LIN {X 0,Y 312.499,Z 218.851,A -85,B 0,C 180,E1 -15693.692,E2 -15693.692} C_VEL
LIN {X 0,Y 312.5,Z 218.867,A -85,B 0,C 180,E1 -15697.39,E2 -15697.39} C_VEL
LIN {X 0,Y 312.472,Z 218.863,A -85,B 0,C 180,E1 -15700.713,E2 -15700.713} C_VEL
LIN {X 0,Y 312.435,Z 218.864,A -85,B 0,C 180,E1 -15704.214,E2 -15704.214} C_VEL
LIN {X 0,Y 312.468,Z 218.877,A -85,B 0,C 180,E1 -15707.923,E2 -15707.923} C_VEL
LIN {X 0,Y 312.464,Z 218.86,A -85,B 0,C 180,E1 -15710.972,E2 -15710.972} C_VEL
LIN {X 0,Y 312.52,Z 218.86,A -85,B 0,C 180,E1 -15714.224,E2 -15714.224} C_VEL
LIN {X 0,Y 312.492,Z 218.871,A -85,B 0,C 180,E1 -15717.338,E2 -15717.338} C_VEL
LIN {X 0,Y 312.5,Z 218.867,A -85,B 0,C 180,E1 -15721.296,E2 -15721.296} C_VEL
LIN {X 0,Y 312.541,Z 218.857,A -85,B 0,C 180,E1 -15724.712,E2 -15724.712} C_VEL
LIN {X 0,Y 312.52,Z 218.87,A -85,B 0,C 180,E1 -15728.916,E2 -15728.916} C_VEL
LIN {X 0,Y 312.56,Z 218.863,A -85,B 0,C 180,E1 -15731.261,E2 -15731.261} C_VEL
LIN {X 0,Y 313.478,Z 221.573,A -85,B 0,C 180,E1 -15731.502,E2 -15731.502} C_VEL
LIN {X 0,Y 315.576,Z 224.258,A -85,B 0,C 180,E1 -15731.935,E2 -15731.935} C_VEL
LIN {X 0,Y 317.795,Z 227.6,A -85,B 0,C 180,E1 -15732.4,E2 -15732.4} C_VEL
LIN {X 0,Y 327.062,Z 241.726,A -85,B 0,C 180,E1 -15734.245,E2 -15734.245} C_VEL
LIN {X 0,Y 337.694,Z 259.213,A -85,B 0,C 180,E1 -15736.243,E2 -15736.243} C_VEL
LIN {X 0,Y 345.227,Z 274.119,A -85,B 0,C 180,E1 -15737.624,E2 -15737.624} C_VEL
LIN {X 0,Y 346.756,Z 277.46,A -85,B 0,C 180,E1 -15737.905,E2 -15737.905} C_VEL
LIN {X 0,Y 340.957,Z 418.481,A -85,B 0,C 180,E1 -15740.961,E2 -15740.961} C_VEL
LIN {X 0,Y 339.666,Z 435.003,A -85,B 0,C 180,E1 -15741.526,E2 -15741.526} C_VEL
LIN {X 0,Y 337.912,Z 451.285,A -85,B 0,C 180,E1 -15742.309,E2 -15742.309} C_VEL
LIN {X 0,Y 335.803,Z 467.163,A -85,B 0,C 180,E1 -15743.318,E2 -15743.318} C_VEL
LIN {X 0,Y 333.363,Z 482.624,A -85,B 0,C 180,E1 -15744.559,E2 -15744.559} C_VEL
LIN {X 0,Y 330.649,Z 497.357,A -85,B 0,C 180,E1 -15746.014,E2 -15746.014} C_VEL
LIN {X 0,Y 327.769,Z 511.318,A -85,B 0,C 180,E1 -15747.699,E2 -15747.699} C_VEL
LIN {X 0,Y 325.107,Z 523.063,A -85,B 0,C 180,E1 -15749.384,E2 -15749.384} C_VEL
LIN {X 0,Y 322.619,Z 534.15,A -85,B 0,C 180,E1 -15751.251,E2 -15751.251} C_VEL
LIN {X 0,Y 319.935,Z 545.24,A -85,B 0,C 180,E1 -15753.466,E2 -15753.466} C_VEL
LIN {X 0,Y 317.551,Z 555.075,A -85,B 0,C 180,E1 -15755.813,E2 -15755.813} C_VEL
LIN {X 0,Y 315.438,Z 563.917,A -85,B 0,C 180,E1 -15758.33,E2 -15758.33} C_VEL
LIN {X 0,Y 313.784,Z 571.615,A -85,B 0,C 180,E1 -15760.978,E2 -15760.978} C_VEL
LIN {X 0,Y 312.529,Z 577.931,A -85,B 0,C 180,E1 -15763.66,E2 -15763.66} C_VEL
LIN {X 0,Y 311.627,Z 583.014,A -85,B 0,C 180,E1 -15766.377,E2 -15766.377} C_VEL
LIN {X 0,Y 311.151,Z 586.089,A -85,B 0,C 180,E1 -15768.437,E2 -15768.437} C_VEL
LIN {X 0,Y 310.646,Z 589.194,A -85,B 0,C 180,E1 -15771.224,E2 -15771.224} C_VEL
LIN {X 0,Y 310.372,Z 591.225,A -85,B 0,C 180,E1 -15774.056,E2 -15774.056} C_VEL
LIN {X 0,Y 310.342,Z 592.031,A -85,B 0,C 180,E1 -15776.933,E2 -15776.933} C_VEL
LIN {X 0,Y 310.449,Z 591.683,A -85,B 0,C 180,E1 -15779.873,E2 -15779.873} C_VEL
LIN {X 0,Y 310.685,Z 590.096,A -85,B 0,C 180,E1 -15782.884,E2 -15782.884} C_VEL
LIN {X 0,Y 311.169,Z 587.504,A -85,B 0,C 180,E1 -15785.6,E2 -15785.6} C_VEL
LIN {X 0,Y 311.823,Z 584.455,A -85,B 0,C 180,E1 -15787.921,E2 -15787.921} C_VEL
LIN {X 0,Y 312.836,Z 579.795,A -85,B 0,C 180,E1 -15790.621,E2 -15790.621} C_VEL
LIN {X 0,Y 312.66,Z 577.864,A -85,B 0,C 180,E1 -15791.643,E2 -15791.643} C_VEL
LIN {X 0,Y 310.678,Z 574.56,A -85,B 0,C 180,E1 -15793.323,E2 -15793.323} C_VEL
LIN {X 0,Y 308.852,Z 570.931,A -85,B 0,C 180,E1 -15794.998,E2 -15794.998} C_VEL
LIN {X 0,Y 308.926,Z 568.371,A -85,B 0,C 180,E1 -15795.991,E2 -15795.991} C_VEL
LIN {X 0,Y 311.415,Z 559.856,A -85,B 0,C 180,E1 -15798.719,E2 -15798.719} C_VEL
LIN {X 0,Y 314.117,Z 550.493,A -85,B 0,C 180,E1 -15801.209,E2 -15801.209} C_VEL
LIN {X 0,Y 317.096,Z 540.388,A -85,B 0,C 180,E1 -15803.46,E2 -15803.46} C_VEL
LIN {X 0,Y 320.339,Z 528.936,A -85,B 0,C 180,E1 -15805.596,E2 -15805.596} C_VEL
LIN {X 0,Y 323.619,Z 516.635,A -85,B 0,C 180,E1 -15807.515,E2 -15807.515} C_VEL
LIN {X 0,Y 327.011,Z 503.039,A -85,B 0,C 180,E1 -15809.281,E2 -15809.281} C_VEL
LIN {X 0,Y 330.189,Z 489.128,A -85,B 0,C 180,E1 -15810.773,E2 -15810.773} C_VEL
LIN {X 0,Y 333.066,Z 474.376,A -85,B 0,C 180,E1 -15812.082,E2 -15812.082} C_VEL
LIN {X 0,Y 335.817,Z 458.032,A -85,B 0,C 180,E1 -15813.218,E2 -15813.218} C_VEL
LIN {X 0,Y 337.97,Z 441.536,A -85,B 0,C 180,E1 -15814.106,E2 -15814.106} C_VEL
LIN {X 0,Y 339.513,Z 426.232,A -85,B 0,C 180,E1 -15814.707,E2 -15814.707} C_VEL
LIN {X 0,Y 340.683,Z 408.213,A -85,B 0,C 180,E1 -15815.189,E2 -15815.189} C_VEL
LIN {X 0,Y 346.82,Z 283.058,A -85,B 0,C 180,E1 -15817.956,E2 -15817.956} C_VEL
LIN {X 0,Y 340.843,Z 271.151,A -85,B 0,C 180,E1 -15819.35,E2 -15819.35} C_VEL
LIN {X 0,Y 335.608,Z 261.937,A -85,B 0,C 180,E1 -15820.612,E2 -15820.612} C_VEL
LIN {X 0,Y 328.374,Z 250.883,A -85,B 0,C 180,E1 -15822.45,E2 -15822.45} C_VEL
LIN {X 0,Y 322.618,Z 242.69,A -85,B 0,C 180,E1 -15824.028,E2 -15824.028} C_VEL
LIN {X 0,Y 320.08,Z 239.215,A -85,B 0,C 180,E1 -15824.762,E2 -15824.762} C_VEL
LIN {X 0,Y 316.654,Z 234.675,A -85,B 0,C 180,E1 -15825.796,E2 -15825.796} C_VEL
LIN {X 0,Y 314.086,Z 231.193,A -85,B 0,C 180,E1 -15826.617,E2 -15826.617} C_VEL
LIN {X 0,Y 313.539,Z 230.399,A -85,B 0,C 180,E1 -15826.799,E2 -15826.799} C_VEL
LIN {X 0,Y 311.036,Z 227.861,A -85,B 0,C 180,E1 -15827.604,E2 -15827.604} C_VEL
LIN {X 0,Y 309.624,Z 225.269,A -85,B 0,C 180,E1 -15828.129,E2 -15828.129} C_VEL
LIN {X 0,Y 307.205,Z 223.361,A -85,B 0,C 180,E1 -15828.953,E2 -15828.953} C_VEL
LIN {X 0,Y 305.962,Z 221.144,A -85,B 0,C 180,E1 -15829.452,E2 -15829.452} C_VEL
LIN {X 0,Y 305.646,Z 219.722,A -85,B 0,C 180,E1 -15829.65,E2 -15829.65} C_VEL
LIN {X 0,Y 305.844,Z 219.698,A -85,B 0,C 180,E1 -15833.402,E2 -15833.402} C_VEL
LIN {X 0,Y 305.958,Z 219.681,A -85,B 0,C 180,E1 -15838.683,E2 -15838.683} C_VEL
LIN {X 0,Y 305.958,Z 219.681,A -85,B 0,C 180,E1 -15841.316,E2 -15841.316} C_VEL
LIN {X 0,Y 305.677,Z 219.717,A -85,B 0,C 180,E1 -15845.276,E2 -15845.276} C_VEL
LIN {X 0,Y 305.767,Z 219.705,A -85,B 0,C 180,E1 -15847.926,E2 -15847.926} C_VEL
LIN {X 0,Y 305.601,Z 219.731,A -85,B 0,C 180,E1 -15851.945,E2 -15851.945} C_VEL
LIN {X 0,Y 305.612,Z 219.729,A -85,B 0,C 180,E1 -15855.013,E2 -15855.013} C_VEL
LIN {X 0,Y 305.521,Z 219.734,A -85,B 0,C 180,E1 -15858.786,E2 -15858.786} C_VEL
LIN {X 0,Y 305.491,Z 219.745,A -85,B 0,C 180,E1 -15863.038,E2 -15863.038} C_VEL
LIN {X 0,Y 305.535,Z 219.737,A -85,B 0,C 180,E1 -15866.219,E2 -15866.219} C_VEL
LIN {X 0,Y 305.484,Z 219.742,A -85,B 0,C 180,E1 -15869.043,E2 -15869.043} C_VEL
LIN {X 0,Y 305.468,Z 219.746,A -85,B 0,C 180,E1 -15873.516,E2 -15873.516} C_VEL
LIN {X 0,Y 305.513,Z 219.832,A -85,B 0,C 180,E1 -15875.788,E2 -15875.788} C_VEL
LIN {X 0,Y 306.147,Z 222.012,A -85,B 0,C 180,E1 -15876.645,E2 -15876.645} C_VEL
LIN {X 0,Y 307.4,Z 224.338,A -85,B 0,C 180,E1 -15877.703,E2 -15877.703} C_VEL
LIN {X 0,Y 309.267,Z 227.241,A -85,B 0,C 180,E1 -15878.492,E2 -15878.492} C_VEL
LIN {X 0,Y 313.704,Z 233.179,A -85,B 0,C 180,E1 -15880,E2 -15880} C_VEL
LIN {X 0,Y 317.317,Z 238.242,A -85,B 0,C 180,E1 -15881.152,E2 -15881.152} C_VEL
LIN {X 0,Y 321.927,Z 245.16,A -85,B 0,C 180,E1 -15882.542,E2 -15882.542} C_VEL
LIN {X 0,Y 327.398,Z 253.587,A -85,B 0,C 180,E1 -15884.077,E2 -15884.077} C_VEL
LIN {X 0,Y 335.467,Z 267.441,A -85,B 0,C 180,E1 -15886.18,E2 -15886.18} C_VEL
LIN {X 0,Y 343.362,Z 283.038,A -85,B 0,C 180,E1 -15888.1,E2 -15888.1} C_VEL
LIN {X 0,Y 346.607,Z 290.135,A -85,B 0,C 180,E1 -15888.859,E2 -15888.859} C_VEL
LIN {X 0,Y 339.477,Z 434.794,A -85,B 0,C 180,E1 -15892.086,E2 -15892.086} C_VEL
LIN {X 0,Y 337.698,Z 452.307,A -85,B 0,C 180,E1 -15892.684,E2 -15892.684} C_VEL
LIN {X 0,Y 335.539,Z 467.974,A -85,B 0,C 180,E1 -15893.44,E2 -15893.44} C_VEL
LIN {X 0,Y 333.18,Z 482.54,A -85,B 0,C 180,E1 -15894.356,E2 -15894.356} C_VEL
LIN {X 0,Y 330.305,Z 497.201,A -85,B 0,C 180,E1 -15895.491,E2 -15895.491} C_VEL
LIN {X 0,Y 326.965,Z 512.316,A -85,B 0,C 180,E1 -15896.959,E2 -15896.959} C_VEL
LIN {X 0,Y 323.553,Z 526.015,A -85,B 0,C 180,E1 -15898.578,E2 -15898.578} C_VEL
LIN {X 0,Y 320.202,Z 538.841,A -85,B 0,C 180,E1 -15900.404,E2 -15900.404} C_VEL
LIN {X 0,Y 316.687,Z 551.596,A -85,B 0,C 180,E1 -15902.583,E2 -15902.583} C_VEL
LIN {X 0,Y 313.643,Z 562.468,A -85,B 0,C 180,E1 -15904.8,E2 -15904.8} C_VEL
LIN {X 0,Y 310.675,Z 572.968,A -85,B 0,C 180,E1 -15907.381,E2 -15907.381} C_VEL
LIN {X 0,Y 308.394,Z 581.802,A -85,B 0,C 180,E1 -15910.009,E2 -15910.009} C_VEL
LIN {X 0,Y 306.554,Z 589.228,A -85,B 0,C 180,E1 -15912.658,E2 -15912.658} C_VEL
LIN {X 0,Y 305.257,Z 595.376,A -85,B 0,C 180,E1 -15915.327,E2 -15915.327} C_VEL
LIN {X 0,Y 304.351,Z 600.312,A -85,B 0,C 180,E1 -15918.002,E2 -15918.002} C_VEL
LIN {X 0,Y 303.818,Z 604.233,A -85,B 0,C 180,E1 -15920.678,E2 -15920.678} C_VEL
LIN {X 0,Y 303.618,Z 607.016,A -85,B 0,C 180,E1 -15923.351,E2 -15923.351} C_VEL
LIN {X 0,Y 303.566,Z 608.889,A -85,B 0,C 180,E1 -15926.014,E2 -15926.014} C_VEL
LIN {X 0,Y 303.574,Z 609.683,A -85,B 0,C 180,E1 -15928.67,E2 -15928.67} C_VEL
LIN {X 0,Y 303.577,Z 609.585,A -85,B 0,C 180,E1 -15931.323,E2 -15931.323} C_VEL
LIN {X 0,Y 303.597,Z 608.406,A -85,B 0,C 180,E1 -15933.979,E2 -15933.979} C_VEL
LIN {X 0,Y 303.614,Z 606.305,A -85,B 0,C 180,E1 -15936.643,E2 -15936.643} C_VEL
LIN {X 0,Y 303.81,Z 603.085,A -85,B 0,C 180,E1 -15939.315,E2 -15939.315} C_VEL
LIN {X 0,Y 304.3,Z 598.835,A -85,B 0,C 180,E1 -15941.993,E2 -15941.993} C_VEL
LIN {X 0,Y 305.255,Z 593.195,A -85,B 0,C 180,E1 -15944.767,E2 -15944.767} C_VEL
LIN {X 0,Y 306.38,Z 586.699,A -85,B 0,C 180,E1 -15947.346,E2 -15947.346} C_VEL
LIN {X 0,Y 308.146,Z 578.641,A -85,B 0,C 180,E1 -15950.001,E2 -15950.001} C_VEL
LIN {X 0,Y 310.378,Z 568.998,A -85,B 0,C 180,E1 -15952.636,E2 -15952.636} C_VEL
LIN {X 0,Y 312.827,Z 558.961,A -85,B 0,C 180,E1 -15954.908,E2 -15954.908} C_VEL
LIN {X 0,Y 315.406,Z 548.282,A -85,B 0,C 180,E1 -15956.965,E2 -15956.965} C_VEL
LIN {X 0,Y 318.263,Z 536.565,A -85,B 0,C 180,E1 -15958.88,E2 -15958.88} C_VEL
LIN {X 0,Y 321.357,Z 522.943,A -85,B 0,C 180,E1 -15960.739,E2 -15960.739} C_VEL
LIN {X 0,Y 324.371,Z 508.574,A -85,B 0,C 180,E1 -15962.352,E2 -15962.352} C_VEL
LIN {X 0,Y 326.997,Z 495.083,A -85,B 0,C 180,E1 -15963.598,E2 -15963.598} C_VEL
LIN {X 0,Y 329.585,Z 479.543,A -85,B 0,C 180,E1 -15964.774,E2 -15964.774} C_VEL
LIN {X 0,Y 331.779,Z 463.658,A -85,B 0,C 180,E1 -15965.717,E2 -15965.717} C_VEL
LIN {X 0,Y 333.636,Z 447.478,A -85,B 0,C 180,E1 -15966.412,E2 -15966.412} C_VEL
LIN {X 0,Y 334.912,Z 430.449,A -85,B 0,C 180,E1 -15966.925,E2 -15966.925} C_VEL
LIN {X 0,Y 340.879,Z 287.591,A -85,B 0,C 180,E1 -15970.057,E2 -15970.057} C_VEL
LIN {X 0,Y 332.472,Z 270.051,A -85,B 0,C 180,E1 -15971.661,E2 -15971.661} C_VEL
LIN {X 0,Y 323.852,Z 253.685,A -85,B 0,C 180,E1 -15973.377,E2 -15973.377} C_VEL
LIN {X 0,Y 314.411,Z 237.36,A -85,B 0,C 180,E1 -15975.347,E2 -15975.347} C_VEL
LIN {X 0,Y 308.193,Z 227.192,A -85,B 0,C 180,E1 -15976.723,E2 -15976.723} C_VEL
LIN {X 0,Y 305.431,Z 219.739,A -85,B 0,C 180,E1 -15978.785,E2 -15978.785} C_VEL
LIN {X 0,Y 305.485,Z 219.746,A -85,B 0,C 180,E1 -15981.6,E2 -15981.6} C_VEL
LIN {X 0,Y 305.438,Z 219.745,A -85,B 0,C 180,E1 -15984.884,E2 -15984.884} C_VEL
LIN {X 0,Y 305.423,Z 219.73,A -85,B 0,C 180,E1 -15988.354,E2 -15988.354} C_VEL
LIN {X 0,Y 305.486,Z 219.747,A -85,B 0,C 180,E1 -15991.111,E2 -15991.111} C_VEL
LIN {X 0,Y 305.539,Z 219.712,A -85,B 0,C 180,E1 -15994.086,E2 -15994.086} C_VEL
LIN {X 0,Y 305.508,Z 219.728,A -85,B 0,C 180,E1 -15998.404,E2 -15998.404} C_VEL
LIN {X 0,Y 305.565,Z 219.707,A -85,B 0,C 180,E1 -16001.217,E2 -16001.217} C_VEL
LIN {X 0,Y 305.62,Z 219.718,A -85,B 0,C 180,E1 -16005.348,E2 -16005.348} C_VEL
LIN {X 0,Y 305.61,Z 219.701,A -85,B 0,C 180,E1 -16009.399,E2 -16009.399} C_VEL
LIN {X 0,Y 305.78,Z 219.708,A -85,B 0,C 180,E1 -16012.074,E2 -16012.074} C_VEL
LIN {X 0,Y 305.659,Z 219.692,A -85,B 0,C 180,E1 -16014.724,E2 -16014.724} C_VEL
LIN {X 0,Y 305.929,Z 219.67,A -85,B 0,C 180,E1 -16018.684,E2 -16018.684} C_VEL
LIN {X 0,Y 305.929,Z 219.688,A -85,B 0,C 180,E1 -16021.317,E2 -16021.317} C_VEL
LIN {X 0,Y 305.813,Z 219.694,A -85,B 0,C 180,E1 -16026.599,E2 -16026.599} C_VEL
LIN {X 0,Y 305.676,Z 219.715,A -85,B 0,C 180,E1 -16029.262,E2 -16029.262} C_VEL
LIN {X 0,Y 305.56,Z 219.719,A -85,B 0,C 180,E1 -16033.298,E2 -16033.298} C_VEL
LIN {X 0,Y 305.567,Z 219.733,A -85,B 0,C 180,E1 -16036.022,E2 -16036.022} C_VEL
LIN {X 0,Y 305.552,Z 219.71,A -85,B 0,C 180,E1 -16039.447,E2 -16039.447} C_VEL
LIN {X 0,Y 305.466,Z 219.744,A -85,B 0,C 180,E1 -16043.044,E2 -16043.044} C_VEL
LIN {X 0,Y 305.502,Z 219.716,A -85,B 0,C 180,E1 -16046.221,E2 -16046.221} C_VEL
LIN {X 0,Y 305.473,Z 219.746,A -85,B 0,C 180,E1 -16049.053,E2 -16049.053} C_VEL
LIN {X 0,Y 305.444,Z 219.728,A -85,B 0,C 180,E1 -16053.52,E2 -16053.52} C_VEL
LIN {X 0,Y 305.453,Z 219.747,A -85,B 0,C 180,E1 -16056.743,E2 -16056.743} C_VEL
LIN {X 0,Y 305.437,Z 219.737,A -85,B 0,C 180,E1 -16060.603,E2 -16060.603} C_VEL
LIN {X 0,Y 305.409,Z 219.746,A -85,B 0,C 180,E1 -16063.659,E2 -16063.659} C_VEL
LIN {X 0,Y 305.439,Z 219.749,A -85,B 0,C 180,E1 -16067.419,E2 -16067.419} C_VEL
LIN {X 0,Y 305.444,Z 219.736,A -85,B 0,C 180,E1 -16069.896,E2 -16069.896} C_VEL
LIN {X 0,Y 305.468,Z 219.747,A -85,B 0,C 180,E1 -16073.636,E2 -16073.636} C_VEL
LIN {X 0,Y 305.455,Z 219.737,A -85,B 0,C 180,E1 -16076.487,E2 -16076.487} C_VEL
LIN {X 0,Y 305.422,Z 219.741,A -85,B 0,C 180,E1 -16079.591,E2 -16079.591} C_VEL
LIN {X 0,Y 305.451,Z 219.749,A -85,B 0,C 180,E1 -16082.606,E2 -16082.606} C_VEL
LIN {X 0,Y 305.477,Z 219.745,A -85,B 0,C 180,E1 -16085.541,E2 -16085.541} C_VEL
LIN {X 0,Y 305.48,Z 219.744,A -85,B 0,C 180,E1 -16089.817,E2 -16089.817} C_VEL
LIN {X 0,Y 305.498,Z 219.886,A -85,B 0,C 180,E1 -16090.078,E2 -16090.078} C_VEL
LIN {X 0,Y 306.586,Z 222.695,A -85,B 0,C 180,E1 -16090.363,E2 -16090.363} C_VEL
LIN {X 0,Y 308.505,Z 224.931,A -85,B 0,C 180,E1 -16090.769,E2 -16090.769} C_VEL
LIN {X 0,Y 310.705,Z 228.389,A -85,B 0,C 180,E1 -16091.256,E2 -16091.256} C_VEL
LIN {X 0,Y 321.632,Z 244.769,A -85,B 0,C 180,E1 -16093.527,E2 -16093.527} C_VEL
LIN {X 0,Y 333.46,Z 264.376,A -85,B 0,C 180,E1 -16095.815,E2 -16095.815} C_VEL
LIN {X 0,Y 340.899,Z 279.517,A -85,B 0,C 180,E1 -16097.224,E2 -16097.224} C_VEL
LIN {X 0,Y 337.693,Z 354.656,A -85,B 0,C 180,E1 -16098.857,E2 -16098.857} C_VEL
LIN {X 0,Y 335.026,Z 419.243,A -85,B 0,C 180,E1 -16100.308,E2 -16100.308} C_VEL
LIN {X 0,Y 333.599,Z 436.411,A -85,B 0,C 180,E1 -16100.912,E2 -16100.912} C_VEL
LIN {X 0,Y 331.816,Z 452.331,A -85,B 0,C 180,E1 -16101.707,E2 -16101.707} C_VEL
LIN {X 0,Y 329.645,Z 468.024,A -85,B 0,C 180,E1 -16102.731,E2 -16102.731} C_VEL
LIN {X 0,Y 327.126,Z 483.37,A -85,B 0,C 180,E1 -16103.991,E2 -16103.991} C_VEL
LIN {X 0,Y 324.303,Z 498.093,A -85,B 0,C 180,E1 -16105.475,E2 -16105.475} C_VEL
LIN {X 0,Y 321.357,Z 511.934,A -85,B 0,C 180,E1 -16107.183,E2 -16107.183} C_VEL
LIN {X 0,Y 318.351,Z 524.612,A -85,B 0,C 180,E1 -16109.054,E2 -16109.054} C_VEL
LIN {X 0,Y 315.343,Z 537.148,A -85,B 0,C 180,E1 -16111.28,E2 -16111.28} C_VEL
LIN {X 0,Y 312.658,Z 547.851,A -85,B 0,C 180,E1 -16113.547,E2 -16113.547} C_VEL
LIN {X 0,Y 310.312,Z 557.25,A -85,B 0,C 180,E1 -16115.909,E2 -16115.909} C_VEL
LIN {X 0,Y 308.21,Z 565.862,A -85,B 0,C 180,E1 -16118.526,E2 -16118.526} C_VEL
LIN {X 0,Y 306.554,Z 573.225,A -85,B 0,C 180,E1 -16121.24,E2 -16121.24} C_VEL
LIN {X 0,Y 305.317,Z 579.269,A -85,B 0,C 180,E1 -16123.965,E2 -16123.965} C_VEL
LIN {X 0,Y 304.45,Z 584.167,A -85,B 0,C 180,E1 -16126.774,E2 -16126.774} C_VEL
LIN {X 0,Y 303.941,Z 587.078,A -85,B 0,C 180,E1 -16128.891,E2 -16128.891} C_VEL
LIN {X 0,Y 303.43,Z 590.224,A -85,B 0,C 180,E1 -16132.106,E2 -16132.106} C_VEL
LIN {X 0,Y 303.246,Z 591.912,A -85,B 0,C 180,E1 -16135.328,E2 -16135.328} C_VEL
LIN {X 0,Y 303.291,Z 592.232,A -85,B 0,C 180,E1 -16138.289,E2 -16138.289} C_VEL
LIN {X 0,Y 303.408,Z 591.542,A -85,B 0,C 180,E1 -16141.011,E2 -16141.011} C_VEL
LIN {X 0,Y 303.741,Z 589.758,A -85,B 0,C 180,E1 -16143.735,E2 -16143.735} C_VEL
LIN {X 0,Y 304.427,Z 586.465,A -85,B 0,C 180,E1 -16146.889,E2 -16146.889} C_VEL
LIN {X 0,Y 305.511,Z 581.629,A -85,B 0,C 180,E1 -16150.101,E2 -16150.101} C_VEL
LIN {X 0,Y 306.871,Z 576.163,A -85,B 0,C 180,E1 -16152.872,E2 -16152.872} C_VEL
LIN {X 0,Y 308.779,Z 568.875,A -85,B 0,C 180,E1 -16155.805,E2 -16155.805} C_VEL
LIN {X 0,Y 308.926,Z 568.371,A -85,B 0,C 180,E1 -16155.991,E2 -16155.991} C_VEL
LIN {X 0,Y 309.079,Z 565.759,A -85,B 0,C 180,E1 -16156.975,E2 -16156.975} C_VEL
LIN {X 0,Y 307.714,Z 561.426,A -85,B 0,C 180,E1 -16158.616,E2 -16158.616} C_VEL
LIN {X 0,Y 306.508,Z 556.667,A -85,B 0,C 180,E1 -16160.226,E2 -16160.226} C_VEL
LIN {X 0,Y 306.898,Z 553.389,A -85,B 0,C 180,E1 -16161.142,E2 -16161.142} C_VEL
LIN {X 0,Y 310.07,Z 543.086,A -85,B 0,C 180,E1 -16163.574,E2 -16163.574} C_VEL
LIN {X 0,Y 313.413,Z 531.85,A -85,B 0,C 180,E1 -16165.795,E2 -16165.795} C_VEL
LIN {X 0,Y 316.93,Z 519.443,A -85,B 0,C 180,E1 -16167.845,E2 -16167.845} C_VEL
LIN {X 0,Y 320.298,Z 506.922,A -85,B 0,C 180,E1 -16169.569,E2 -16169.569} C_VEL
LIN {X 0,Y 323.544,Z 493.409,A -85,B 0,C 180,E1 -16171.113,E2 -16171.113} C_VEL
LIN {X 0,Y 326.728,Z 478.327,A -85,B 0,C 180,E1 -16172.538,E2 -16172.538} C_VEL
LIN {X 0,Y 329.672,Z 462.405,A -85,B 0,C 180,E1 -16173.729,E2 -16173.729} C_VEL
LIN {X 0,Y 331.947,Z 446.695,A -85,B 0,C 180,E1 -16174.662,E2 -16174.662} C_VEL
LIN {X 0,Y 333.865,Z 430.084,A -85,B 0,C 180,E1 -16175.385,E2 -16175.385} C_VEL
LIN {X 0,Y 335.222,Z 412.543,A -85,B 0,C 180,E1 -16175.891,E2 -16175.891} C_VEL
LIN {X 0,Y 341.643,Z 285.694,A -85,B 0,C 180,E1 -16178.748,E2 -16178.748} C_VEL
LIN {X 0,Y 336.562,Z 275.405,A -85,B 0,C 180,E1 -16179.984,E2 -16179.984} C_VEL
LIN {X 0,Y 331.57,Z 266.534,A -85,B 0,C 180,E1 -16181.245,E2 -16181.245} C_VEL
LIN {X 0,Y 324.797,Z 256.08,A -85,B 0,C 180,E1 -16183.03,E2 -16183.03} C_VEL
LIN {X 0,Y 318.947,Z 247.567,A -85,B 0,C 180,E1 -16184.702,E2 -16184.702} C_VEL
LIN {X 0,Y 313.781,Z 240.604,A -85,B 0,C 180,E1 -16186.294,E2 -16186.294} C_VEL
LIN {X 0,Y 310.568,Z 236.322,A -85,B 0,C 180,E1 -16187.357,E2 -16187.357} C_VEL
LIN {X 0,Y 307.801,Z 233.016,A -85,B 0,C 180,E1 -16188.308,E2 -16188.308} C_VEL
LIN {X 0,Y 306.8,Z 231.437,A -85,B 0,C 180,E1 -16188.688,E2 -16188.688} C_VEL
LIN {X 0,Y 304.277,Z 228.936,A -85,B 0,C 180,E1 -16189.603,E2 -16189.603} C_VEL
LIN {X 0,Y 302.788,Z 226.206,A -85,B 0,C 180,E1 -16190.227,E2 -16190.227} C_VEL
LIN {X 0,Y 300.365,Z 224.337,A -85,B 0,C 180,E1 -16191.145,E2 -16191.145} C_VEL
LIN {X 0,Y 299.075,Z 222.067,A -85,B 0,C 180,E1 -16191.724,E2 -16191.724} C_VEL
LIN {X 0,Y 298.751,Z 220.58,A -85,B 0,C 180,E1 -16191.97,E2 -16191.97} C_VEL
LIN {X 0,Y 298.658,Z 220.593,A -85,B 0,C 180,E1 -16194.598,E2 -16194.598} C_VEL
LIN {X 0,Y 298.925,Z 220.557,A -85,B 0,C 180,E1 -16198.652,E2 -16198.652} C_VEL
LIN {X 0,Y 298.925,Z 220.557,A -85,B 0,C 180,E1 -16201.347,E2 -16201.347} C_VEL
LIN {X 0,Y 298.646,Z 220.594,A -85,B 0,C 180,E1 -16205.401,E2 -16205.401} C_VEL
LIN {X 0,Y 298.714,Z 220.585,A -85,B 0,C 180,E1 -16208.115,E2 -16208.115} C_VEL
LIN {X 0,Y 298.552,Z 220.607,A -85,B 0,C 180,E1 -16212.231,E2 -16212.231} C_VEL
LIN {X 0,Y 298.552,Z 220.606,A -85,B 0,C 180,E1 -16215.166,E2 -16215.166} C_VEL
LIN {X 0,Y 298.449,Z 220.617,A -85,B 0,C 180,E1 -16219.618,E2 -16219.618} C_VEL
LIN {X 0,Y 298.433,Z 220.621,A -85,B 0,C 180,E1 -16223.599,E2 -16223.599} C_VEL
LIN {X 0,Y 298.491,Z 220.612,A -85,B 0,C 180,E1 -16226.574,E2 -16226.574} C_VEL
LIN {X 0,Y 298.414,Z 220.62,A -85,B 0,C 180,E1 -16229.641,E2 -16229.641} C_VEL
LIN {X 0,Y 298.432,Z 220.64,A -85,B 0,C 180,E1 -16233.601,E2 -16233.601} C_VEL
LIN {X 0,Y 299.611,Z 223.76,A -85,B 0,C 180,E1 -16235.077,E2 -16235.077} C_VEL
LIN {X 0,Y 300.622,Z 224.981,A -85,B 0,C 180,E1 -16235.609,E2 -16235.609} C_VEL
LIN {X 0,Y 302.932,Z 228.411,A -85,B 0,C 180,E1 -16236.565,E2 -16236.565} C_VEL
LIN {X 0,Y 305.322,Z 231.408,A -85,B 0,C 180,E1 -16237.484,E2 -16237.484} C_VEL
LIN {X 0,Y 310.889,Z 239.118,A -85,B 0,C 180,E1 -16239.491,E2 -16239.491} C_VEL
LIN {X 0,Y 314.388,Z 244.11,A -85,B 0,C 180,E1 -16240.649,E2 -16240.649} C_VEL
LIN {X 0,Y 318.591,Z 250.541,A -85,B 0,C 180,E1 -16241.965,E2 -16241.965} C_VEL
LIN {X 0,Y 324.059,Z 259.165,A -85,B 0,C 180,E1 -16243.557,E2 -16243.557} C_VEL
LIN {X 0,Y 331.212,Z 271.637,A -85,B 0,C 180,E1 -16245.496,E2 -16245.496} C_VEL
LIN {X 0,Y 337.899,Z 284.971,A -85,B 0,C 180,E1 -16247.205,E2 -16247.205} C_VEL
LIN {X 0,Y 341.431,Z 292.596,A -85,B 0,C 180,E1 -16248.069,E2 -16248.069} C_VEL
LIN {X 0,Y 336.388,Z 391.224,A -85,B 0,C 180,E1 -16250.277,E2 -16250.277} C_VEL
LIN {X 0,Y 334.139,Z 434.986,A -85,B 0,C 180,E1 -16251.297,E2 -16251.297} C_VEL
LIN {X 0,Y 332.219,Z 452.986,A -85,B 0,C 180,E1 -16251.921,E2 -16251.921} C_VEL
LIN {X 0,Y 329.912,Z 468.908,A -85,B 0,C 180,E1 -16252.712,E2 -16252.712} C_VEL
LIN {X 0,Y 327.468,Z 483.166,A -85,B 0,C 180,E1 -16253.637,E2 -16253.637} C_VEL
LIN {X 0,Y 324.505,Z 497.633,A -85,B 0,C 180,E1 -16254.784,E2 -16254.784} C_VEL
LIN {X 0,Y 320.887,Z 513.248,A -85,B 0,C 180,E1 -16256.331,E2 -16256.331} C_VEL
LIN {X 0,Y 317.201,Z 527.425,A -85,B 0,C 180,E1 -16258.061,E2 -16258.061} C_VEL
LIN {X 0,Y 314.004,Z 539.005,A -85,B 0,C 180,E1 -16259.76,E2 -16259.76} C_VEL
LIN {X 0,Y 310.513,Z 551.156,A -85,B 0,C 180,E1 -16261.869,E2 -16261.869} C_VEL
LIN {X 0,Y 307.611,Z 561.029,A -85,B 0,C 180,E1 -16263.906,E2 -16263.906} C_VEL
LIN {X 0,Y 304.776,Z 570.473,A -85,B 0,C 180,E1 -16266.198,E2 -16266.198} C_VEL
LIN {X 0,Y 302.143,Z 579.717,A -85,B 0,C 180,E1 -16268.864,E2 -16268.864} C_VEL
LIN {X 0,Y 300.137,Z 587.454,A -85,B 0,C 180,E1 -16271.569,E2 -16271.569} C_VEL
LIN {X 0,Y 298.618,Z 593.833,A -85,B 0,C 180,E1 -16274.294,E2 -16274.294} C_VEL
LIN {X 0,Y 297.562,Z 599.092,A -85,B 0,C 180,E1 -16277.031,E2 -16277.031} C_VEL
LIN {X 0,Y 296.737,Z 604.081,A -85,B 0,C 180,E1 -16280.454,E2 -16280.454} C_VEL
LIN {X 0,Y 296.533,Z 606.85,A -85,B 0,C 180,E1 -16283.191,E2 -16283.191} C_VEL
LIN {X 0,Y 296.468,Z 608.701,A -85,B 0,C 180,E1 -16285.919,E2 -16285.919} C_VEL
LIN {X 0,Y 296.493,Z 609.483,A -85,B 0,C 180,E1 -16288.639,E2 -16288.639} C_VEL
LIN {X 0,Y 296.496,Z 609.362,A -85,B 0,C 180,E1 -16291.355,E2 -16291.355} C_VEL
LIN {X 0,Y 296.494,Z 608.168,A -85,B 0,C 180,E1 -16294.074,E2 -16294.074} C_VEL
LIN {X 0,Y 296.529,Z 606.041,A -85,B 0,C 180,E1 -16296.802,E2 -16296.802} C_VEL
LIN {X 0,Y 296.828,Z 601.879,A -85,B 0,C 180,E1 -16300.225,E2 -16300.225} C_VEL
LIN {X 0,Y 297.719,Z 595.981,A -85,B 0,C 180,E1 -16303.65,E2 -16303.65} C_VEL
LIN {X 0,Y 298.772,Z 589.865,A -85,B 0,C 180,E1 -16306.392,E2 -16306.392} C_VEL
LIN {X 0,Y 300.441,Z 582.475,A -85,B 0,C 180,E1 -16309.112,E2 -16309.112} C_VEL
LIN {X 0,Y 302.451,Z 573.611,A -85,B 0,C 180,E1 -16311.822,E2 -16311.822} C_VEL
LIN {X 0,Y 305.149,Z 563.025,A -85,B 0,C 180,E1 -16314.487,E2 -16314.487} C_VEL
LIN {X 0,Y 307.953,Z 552,A -85,B 0,C 180,E1 -16316.786,E2 -16316.786} C_VEL
LIN {X 0,Y 310.656,Z 540.988,A -85,B 0,C 180,E1 -16318.729,E2 -16318.729} C_VEL
LIN {X 0,Y 313.754,Z 528.221,A -85,B 0,C 180,E1 -16320.632,E2 -16320.632} C_VEL
LIN {X 0,Y 317.044,Z 513.888,A -85,B 0,C 180,E1 -16322.397,E2 -16322.397} C_VEL
LIN {X 0,Y 320.042,Z 499.337,A -85,B 0,C 180,E1 -16323.859,E2 -16323.859} C_VEL
LIN {X 0,Y 322.872,Z 483.699,A -85,B 0,C 180,E1 -16325.127,E2 -16325.127} C_VEL
LIN {X 0,Y 325.286,Z 467.588,A -85,B 0,C 180,E1 -16326.159,E2 -16326.159} C_VEL
LIN {X 0,Y 327.235,Z 451.972,A -85,B 0,C 180,E1 -16326.913,E2 -16326.913} C_VEL
LIN {X 0,Y 328.762,Z 435.22,A -85,B 0,C 180,E1 -16327.491,E2 -16327.491} C_VEL
LIN {X 0,Y 335.163,Z 290.859,A -85,B 0,C 180,E1 -16330.707,E2 -16330.707} C_VEL
LIN {X 0,Y 334.81,Z 289.109,A -85,B 0,C 180,E1 -16330.803,E2 -16330.803} C_VEL
LIN {X 0,Y 325.695,Z 270.313,A -85,B 0,C 180,E1 -16332.61,E2 -16332.61} C_VEL
LIN {X 0,Y 317.461,Z 254.826,A -85,B 0,C 180,E1 -16334.312,E2 -16334.312} C_VEL
LIN {X 0,Y 309.74,Z 241.556,A -85,B 0,C 180,E1 -16335.983,E2 -16335.983} C_VEL
LIN {X 0,Y 300.741,Z 226.876,A -85,B 0,C 180,E1 -16338.073,E2 -16338.073} C_VEL
LIN {X 0,Y 298.403,Z 220.615,A -85,B 0,C 180,E1 -16339.91,E2 -16339.91} C_VEL
LIN {X 0,Y 298.397,Z 220.611,A -85,B 0,C 180,E1 -16343.928,E2 -16343.928} C_VEL
LIN {X 0,Y 298.368,Z 220.608,A -85,B 0,C 180,E1 -16347.982,E2 -16347.982} C_VEL
LIN {X 0,Y 298.422,Z 220.617,A -85,B 0,C 180,E1 -16351.901,E2 -16351.901} C_VEL
LIN {X 0,Y 298.46,Z 220.601,A -85,B 0,C 180,E1 -16354.922,E2 -16354.922} C_VEL
LIN {X 0,Y 298.428,Z 220.62,A -85,B 0,C 180,E1 -16357.865,E2 -16357.865} C_VEL
LIN {X 0,Y 298.531,Z 220.579,A -85,B 0,C 180,E1 -16360.757,E2 -16360.757} C_VEL
LIN {X 0,Y 298.565,Z 220.6,A -85,B 0,C 180,E1 -16364.994,E2 -16364.994} C_VEL
LIN {X 0,Y 298.566,Z 220.574,A -85,B 0,C 180,E1 -16369.146,E2 -16369.146} C_VEL
LIN {X 0,Y 298.727,Z 220.586,A -85,B 0,C 180,E1 -16371.886,E2 -16371.886} C_VEL
LIN {X 0,Y 298.63,Z 220.568,A -85,B 0,C 180,E1 -16374.599,E2 -16374.599} C_VEL
LIN {X 0,Y 298.896,Z 220.545,A -85,B 0,C 180,E1 -16378.653,E2 -16378.653} C_VEL
LIN {X 0,Y 298.895,Z 220.565,A -85,B 0,C 180,E1 -16381.348,E2 -16381.348} C_VEL
LIN {X 0,Y 298.759,Z 220.574,A -85,B 0,C 180,E1 -16386.755,E2 -16386.755} C_VEL
LIN {X 0,Y 298.608,Z 220.594,A -85,B 0,C 180,E1 -16389.484,E2 -16389.484} C_VEL
LIN {X 0,Y 298.524,Z 220.601,A -85,B 0,C 180,E1 -16393.617,E2 -16393.617} C_VEL
LIN {X 0,Y 298.523,Z 220.605,A -85,B 0,C 180,E1 -16396.411,E2 -16396.411} C_VEL
LIN {X 0,Y 298.487,Z 220.591,A -85,B 0,C 180,E1 -16399.657,E2 -16399.657} C_VEL
LIN {X 0,Y 298.433,Z 220.619,A -85,B 0,C 180,E1 -16403.6,E2 -16403.6} C_VEL
LIN {X 0,Y 298.463,Z 220.594,A -85,B 0,C 180,E1 -16406.578,E2 -16406.578} C_VEL
LIN {X 0,Y 298.399,Z 220.627,A -85,B 0,C 180,E1 -16409.644,E2 -16409.644} C_VEL
LIN {X 0,Y 298.374,Z 220.605,A -85,B 0,C 180,E1 -16412.804,E2 -16412.804} C_VEL
LIN {X 0,Y 298.425,Z 220.622,A -85,B 0,C 180,E1 -16416.81,E2 -16416.81} C_VEL
LIN {X 0,Y 298.37,Z 220.625,A -85,B 0,C 180,E1 -16421.091,E2 -16421.091} C_VEL
LIN {X 0,Y 298.383,Z 220.627,A -85,B 0,C 180,E1 -16423.107,E2 -16423.107} C_VEL
LIN {X 0,Y 298.389,Z 220.624,A -85,B 0,C 180,E1 -16426.925,E2 -16426.925} C_VEL
LIN {X 0,Y 298.378,Z 220.614,A -85,B 0,C 180,E1 -16431.014,E2 -16431.014} C_VEL
LIN {X 0,Y 298.406,Z 220.621,A -85,B 0,C 180,E1 -16433.934,E2 -16433.934} C_VEL
LIN {X 0,Y 298.383,Z 220.629,A -85,B 0,C 180,E1 -16437.204,E2 -16437.204} C_VEL
LIN {X 0,Y 298.395,Z 220.616,A -85,B 0,C 180,E1 -16440.629,E2 -16440.629} C_VEL
LIN {X 0,Y 298.438,Z 220.615,A -85,B 0,C 180,E1 -16444.924,E2 -16444.924} C_VEL
LIN {X 0,Y 298.419,Z 220.623,A -85,B 0,C 180,E1 -16448.801,E2 -16448.801} C_VEL
LIN {X 0,Y 299.406,Z 223.471,A -85,B 0,C 180,E1 -16449.093,E2 -16449.093} C_VEL
LIN {X 0,Y 301.584,Z 225.989,A -85,B 0,C 180,E1 -16449.582,E2 -16449.582} C_VEL
LIN {X 0,Y 303.603,Z 229.189,A -85,B 0,C 180,E1 -16450.056,E2 -16450.056} C_VEL
LIN {X 0,Y 304.886,Z 230.986,A -85,B 0,C 180,E1 -16450.343,E2 -16450.343} C_VEL
LIN {X 0,Y 315.219,Z 246.35,A -85,B 0,C 180,E1 -16452.576,E2 -16452.576} C_VEL
LIN {X 0,Y 325.848,Z 263.774,A -85,B 0,C 180,E1 -16454.722,E2 -16454.722} C_VEL
LIN {X 0,Y 330.76,Z 272.757,A -85,B 0,C 180,E1 -16455.681,E2 -16455.681} C_VEL
LIN {X 0,Y 335.257,Z 281.997,A -85,B 0,C 180,E1 -16456.556,E2 -16456.556} C_VEL
LIN {X 0,Y 329.222,Z 418.651,A -85,B 0,C 180,E1 -16459.603,E2 -16459.603} C_VEL
LIN {X 0,Y 327.866,Z 434.931,A -85,B 0,C 180,E1 -16460.168,E2 -16460.168} C_VEL
LIN {X 0,Y 326.084,Z 450.706,A -85,B 0,C 180,E1 -16460.935,E2 -16460.935} C_VEL
LIN {X 0,Y 323.986,Z 465.837,A -85,B 0,C 180,E1 -16461.898,E2 -16461.898} C_VEL
LIN {X 0,Y 321.535,Z 480.75,A -85,B 0,C 180,E1 -16463.099,E2 -16463.099} C_VEL
LIN {X 0,Y 318.829,Z 494.658,A -85,B 0,C 180,E1 -16464.469,E2 -16464.469} C_VEL
LIN {X 0,Y 315.67,Z 509.003,A -85,B 0,C 180,E1 -16466.174,E2 -16466.174} C_VEL
LIN {X 0,Y 312.605,Z 522.163,A -85,B 0,C 180,E1 -16468.071,E2 -16468.071} C_VEL
LIN {X 0,Y 309.577,Z 534.518,A -85,B 0,C 180,E1 -16470.205,E2 -16470.205} C_VEL
LIN {X 0,Y 306.538,Z 546.197,A -85,B 0,C 180,E1 -16472.631,E2 -16472.631} C_VEL
LIN {X 0,Y 303.719,Z 556.842,A -85,B 0,C 180,E1 -16475.314,E2 -16475.314} C_VEL
LIN {X 0,Y 301.415,Z 565.75,A -85,B 0,C 180,E1 -16478.045,E2 -16478.045} C_VEL
LIN {X 0,Y 299.682,Z 573.17,A -85,B 0,C 180,E1 -16480.816,E2 -16480.816} C_VEL
LIN {X 0,Y 298.366,Z 579.316,A -85,B 0,C 180,E1 -16483.627,E2 -16483.627} C_VEL
LIN {X 0,Y 297.432,Z 584.197,A -85,B 0,C 180,E1 -16486.475,E2 -16486.475} C_VEL
LIN {X 0,Y 296.744,Z 587.943,A -85,B 0,C 180,E1 -16489.367,E2 -16489.367} C_VEL
LIN {X 0,Y 296.3,Z 590.631,A -85,B 0,C 180,E1 -16492.322,E2 -16492.322} C_VEL
LIN {X 0,Y 296.138,Z 592.213,A -85,B 0,C 180,E1 -16495.599,E2 -16495.599} C_VEL
LIN {X 0,Y 296.212,Z 592.415,A -85,B 0,C 180,E1 -16498.612,E2 -16498.612} C_VEL
LIN {X 0,Y 296.359,Z 591.6,A -85,B 0,C 180,E1 -16501.45,E2 -16501.45} C_VEL
LIN {X 0,Y 296.782,Z 589.418,A -85,B 0,C 180,E1 -16504.637,E2 -16504.637} C_VEL
LIN {X 0,Y 297.648,Z 585.782,A -85,B 0,C 180,E1 -16507.875,E2 -16507.875} C_VEL
LIN {X 0,Y 298.928,Z 580.526,A -85,B 0,C 180,E1 -16511.205,E2 -16511.205} C_VEL
LIN {X 0,Y 300.376,Z 574.988,A -85,B 0,C 180,E1 -16513.926,E2 -16513.926} C_VEL
LIN {X 0,Y 302.289,Z 568.338,A -85,B 0,C 180,E1 -16516.584,E2 -16516.584} C_VEL
LIN {X 0,Y 304.656,Z 560.733,A -85,B 0,C 180,E1 -16519.071,E2 -16519.071} C_VEL
LIN {X 0,Y 306.898,Z 553.389,A -85,B 0,C 180,E1 -16521.142,E2 -16521.142} C_VEL
LIN {X 0,Y 307.346,Z 550.026,A -85,B 0,C 180,E1 -16522.043,E2 -16522.043} C_VEL
LIN {X 0,Y 305.774,Z 538.928,A -85,B 0,C 180,E1 -16525.103,E2 -16525.103} C_VEL
LIN {X 0,Y 306.379,Z 535.091,A -85,B 0,C 180,E1 -16525.935,E2 -16525.935} C_VEL
LIN {X 0,Y 309.873,Z 523.563,A -85,B 0,C 180,E1 -16527.962,E2 -16527.962} C_VEL
LIN {X 0,Y 313.292,Z 511.602,A -85,B 0,C 180,E1 -16529.732,E2 -16529.732} C_VEL
LIN {X 0,Y 316.846,Z 498.03,A -85,B 0,C 180,E1 -16531.416,E2 -16531.416} C_VEL
LIN {X 0,Y 320.275,Z 483.136,A -85,B 0,C 180,E1 -16532.933,E2 -16532.933} C_VEL
LIN {X 0,Y 323.536,Z 466.824,A -85,B 0,C 180,E1 -16534.249,E2 -16534.249} C_VEL
LIN {X 0,Y 326.157,Z 450.52,A -85,B 0,C 180,E1 -16535.275,E2 -16535.275} C_VEL
LIN {X 0,Y 328.186,Z 433.979,A -85,B 0,C 180,E1 -16536.06,E2 -16536.06} C_VEL
LIN {X 0,Y 329.723,Z 416.952,A -85,B 0,C 180,E1 -16536.611,E2 -16536.611} C_VEL
LIN {X 0,Y 336.601,Z 288.377,A -85,B 0,C 180,E1 -16539.553,E2 -16539.553} C_VEL
LIN {X 0,Y 331.397,Z 277.822,A -85,B 0,C 180,E1 -16540.889,E2 -16540.889} C_VEL
LIN {X 0,Y 326.62,Z 269.546,A -85,B 0,C 180,E1 -16542.146,E2 -16542.146} C_VEL
LIN {X 0,Y 319.006,Z 257.9,A -85,B 0,C 180,E1 -16544.28,E2 -16544.28} C_VEL
LIN {X 0,Y 314.175,Z 250.937,A -85,B 0,C 180,E1 -16545.754,E2 -16545.754} C_VEL
LIN {X 0,Y 310.76,Z 246.309,A -85,B 0,C 180,E1 -16546.861,E2 -16546.861} C_VEL
LIN {X 0,Y 307.622,Z 242.15,A -85,B 0,C 180,E1 -16547.935,E2 -16547.935} C_VEL
LIN {X 0,Y 304.751,Z 238.305,A -85,B 0,C 180,E1 -16548.989,E2 -16548.989} C_VEL
LIN {X 0,Y 301.374,Z 234.407,A -85,B 0,C 180,E1 -16550.276,E2 -16550.276} C_VEL
LIN {X 0,Y 300.309,Z 232.581,A -85,B 0,C 180,E1 -16550.73,E2 -16550.73} C_VEL
LIN {X 0,Y 297.727,Z 230.122,A -85,B 0,C 180,E1 -16551.771,E2 -16551.771} C_VEL
LIN {X 0,Y 296.253,Z 227.195,A -85,B 0,C 180,E1 -16552.502,E2 -16552.502} C_VEL
LIN {X 0,Y 293.484,Z 225.376,A -85,B 0,C 180,E1 -16553.727,E2 -16553.727} C_VEL
LIN {X 0,Y 291.979,Z 222.969,A -85,B 0,C 180,E1 -16554.518,E2 -16554.518} C_VEL
LIN {X 0,Y 291.592,Z 221.474,A -85,B 0,C 180,E1 -16554.814,E2 -16554.814} C_VEL
LIN {X 0,Y 291.891,Z 221.433,A -85,B 0,C 180,E1 -16558.62,E2 -16558.62} C_VEL
LIN {X 0,Y 291.891,Z 221.433,A -85,B 0,C 180,E1 -16561.379,E2 -16561.379} C_VEL
LIN {X 0,Y 291.704,Z 221.456,A -85,B 0,C 180,E1 -16566.918,E2 -16566.918} C_VEL
LIN {X 0,Y 291.572,Z 221.472,A -85,B 0,C 180,E1 -16569.713,E2 -16569.713} C_VEL
LIN {X 0,Y 291.518,Z 221.481,A -85,B 0,C 180,E1 -16573.95,E2 -16573.95} C_VEL
LIN {X 0,Y 291.432,Z 221.491,A -85,B 0,C 180,E1 -16576.82,E2 -16576.82} C_VEL
LIN {X 0,Y 291.396,Z 221.497,A -85,B 0,C 180,E1 -16579.841,E2 -16579.841} C_VEL
LIN {X 0,Y 291.387,Z 221.494,A -85,B 0,C 180,E1 -16584.206,E2 -16584.206} C_VEL
LIN {X 0,Y 291.423,Z 221.49,A -85,B 0,C 180,E1 -16587.271,E2 -16587.271} C_VEL
LIN {X 0,Y 291.367,Z 221.637,A -85,B 0,C 180,E1 -16591.136,E2 -16591.136} C_VEL
LIN {X 0,Y 292.154,Z 223.967,A -85,B 0,C 180,E1 -16592.253,E2 -16592.253} C_VEL
LIN {X 0,Y 293.879,Z 226.104,A -85,B 0,C 180,E1 -16593.113,E2 -16593.113} C_VEL
LIN {X 0,Y 294.808,Z 227.01,A -85,B 0,C 180,E1 -16593.547,E2 -16593.547} C_VEL
LIN {X 0,Y 297.216,Z 230.108,A -85,B 0,C 180,E1 -16594.67,E2 -16594.67} C_VEL
LIN {X 0,Y 298.504,Z 231.672,A -85,B 0,C 180,E1 -16595.227,E2 -16595.227} C_VEL
LIN {X 0,Y 300.88,Z 234.974,A -85,B 0,C 180,E1 -16596.219,E2 -16596.219} C_VEL
LIN {X 0,Y 303.588,Z 238.624,A -85,B 0,C 180,E1 -16597.291,E2 -16597.291} C_VEL
LIN {X 0,Y 308.359,Z 245.365,A -85,B 0,C 180,E1 -16599.06,E2 -16599.06} C_VEL
LIN {X 0,Y 312.222,Z 251.094,A -85,B 0,C 180,E1 -16600.376,E2 -16600.376} C_VEL
LIN {X 0,Y 318.374,Z 260.799,A -85,B 0,C 180,E1 -16602.32,E2 -16602.32} C_VEL
LIN {X 0,Y 325.065,Z 272.276,A -85,B 0,C 180,E1 -16604.261,E2 -16604.261} C_VEL
LIN {X 0,Y 331.414,Z 284.508,A -85,B 0,C 180,E1 -16605.98,E2 -16605.98} C_VEL
LIN {X 0,Y 336.382,Z 295.177,A -85,B 0,C 180,E1 -16607.263,E2 -16607.263} C_VEL
LIN {X 0,Y 330.047,Z 414.495,A -85,B 0,C 180,E1 -16609.972,E2 -16609.972} C_VEL
LIN {X 0,Y 328.642,Z 437.594,A -85,B 0,C 180,E1 -16610.561,E2 -16610.561} C_VEL
LIN {X 0,Y 326.736,Z 454.025,A -85,B 0,C 180,E1 -16611.154,E2 -16611.154} C_VEL
LIN {X 0,Y 324.154,Z 471.091,A -85,B 0,C 180,E1 -16612.032,E2 -16612.032} C_VEL
LIN {X 0,Y 321.042,Z 487.763,A -85,B 0,C 180,E1 -16613.18,E2 -16613.18} C_VEL
LIN {X 0,Y 317.646,Z 502.837,A -85,B 0,C 180,E1 -16614.492,E2 -16614.492} C_VEL
LIN {X 0,Y 314.159,Z 516.814,A -85,B 0,C 180,E1 -16615.992,E2 -16615.992} C_VEL
LIN {X 0,Y 310.247,Z 530.961,A -85,B 0,C 180,E1 -16617.834,E2 -16617.834} C_VEL
LIN {X 0,Y 306.746,Z 543.055,A -85,B 0,C 180,E1 -16619.729,E2 -16619.729} C_VEL
LIN {X 0,Y 302.961,Z 555.519,A -85,B 0,C 180,E1 -16622.087,E2 -16622.087} C_VEL
LIN {X 0,Y 299.452,Z 566.656,A -85,B 0,C 180,E1 -16624.637,E2 -16624.637} C_VEL
LIN {X 0,Y 296.411,Z 576.416,A -85,B 0,C 180,E1 -16627.336,E2 -16627.336} C_VEL
LIN {X 0,Y 294.374,Z 583.727,A -85,B 0,C 180,E1 -16629.744,E2 -16629.744} C_VEL
LIN {X 0,Y 292.419,Z 590.718,A -85,B 0,C 180,E1 -16632.514,E2 -16632.514} C_VEL
LIN {X 0,Y 291.033,Z 596.691,A -85,B 0,C 180,E1 -16635.422,E2 -16635.422} C_VEL
LIN {X 0,Y 290.121,Z 601.158,A -85,B 0,C 180,E1 -16638.114,E2 -16638.114} C_VEL
LIN {X 0,Y 289.67,Z 603.936,A -85,B 0,C 180,E1 -16640.219,E2 -16640.219} C_VEL
LIN {X 0,Y 289.445,Z 606.687,A -85,B 0,C 180,E1 -16643.024,E2 -16643.024} C_VEL
LIN {X 0,Y 289.373,Z 608.512,A -85,B 0,C 180,E1 -16645.818,E2 -16645.818} C_VEL
LIN {X 0,Y 289.414,Z 609.283,A -85,B 0,C 180,E1 -16648.605,E2 -16648.605} C_VEL
LIN {X 0,Y 289.417,Z 609.138,A -85,B 0,C 180,E1 -16651.388,E2 -16651.388} C_VEL
LIN {X 0,Y 289.396,Z 607.931,A -85,B 0,C 180,E1 -16654.174,E2 -16654.174} C_VEL
LIN {X 0,Y 289.44,Z 605.776,A -85,B 0,C 180,E1 -16656.97,E2 -16656.97} C_VEL
LIN {X 0,Y 289.664,Z 602.526,A -85,B 0,C 180,E1 -16659.775,E2 -16659.775} C_VEL
LIN {X 0,Y 290.284,Z 598.216,A -85,B 0,C 180,E1 -16662.582,E2 -16662.582} C_VEL
LIN {X 0,Y 291.263,Z 592.752,A -85,B 0,C 180,E1 -16665.388,E2 -16665.388} C_VEL
LIN {X 0,Y 292.644,Z 585.97,A -85,B 0,C 180,E1 -16668.188,E2 -16668.188} C_VEL
LIN {X 0,Y 294.599,Z 577.823,A -85,B 0,C 180,E1 -16670.963,E2 -16670.963} C_VEL
LIN {X 0,Y 297.066,Z 568.08,A -85,B 0,C 180,E1 -16673.71,E2 -16673.71} C_VEL
LIN {X 0,Y 299.821,Z 557.982,A -85,B 0,C 180,E1 -16676.068,E2 -16676.068} C_VEL
LIN {X 0,Y 302.821,Z 546.101,A -85,B 0,C 180,E1 -16678.404,E2 -16678.404} C_VEL
LIN {X 0,Y 306.17,Z 533.117,A -85,B 0,C 180,E1 -16680.517,E2 -16680.517} C_VEL
LIN {X 0,Y 309.384,Z 520.235,A -85,B 0,C 180,E1 -16682.259,E2 -16682.259} C_VEL
LIN {X 0,Y 312.565,Z 505.953,A -85,B 0,C 180,E1 -16683.87,E2 -16683.87} C_VEL
LIN {X 0,Y 315.131,Z 493.195,A -85,B 0,C 180,E1 -16685.043,E2 -16685.043} C_VEL
LIN {X 0,Y 317.892,Z 477.238,A -85,B 0,C 180,E1 -16686.25,E2 -16686.25} C_VEL
LIN {X 0,Y 320.139,Z 461.503,A -85,B 0,C 180,E1 -16687.18,E2 -16687.18} C_VEL
LIN {X 0,Y 322.112,Z 445.05,A -85,B 0,C 180,E1 -16687.884,E2 -16687.884} C_VEL
LIN {X 0,Y 323.407,Z 427.666,A -85,B 0,C 180,E1 -16688.388,E2 -16688.388} C_VEL
LIN {X 0,Y 329.504,Z 292.264,A -85,B 0,C 180,E1 -16691.433,E2 -16691.433} C_VEL
LIN {X 0,Y 320.698,Z 273.981,A -85,B 0,C 180,E1 -16693.232,E2 -16693.232} C_VEL
LIN {X 0,Y 312.551,Z 258.596,A -85,B 0,C 180,E1 -16694.973,E2 -16694.973} C_VEL
LIN {X 0,Y 305.202,Z 245.956,A -85,B 0,C 180,E1 -16696.609,E2 -16696.609} C_VEL
LIN {X 0,Y 296.439,Z 231.624,A -85,B 0,C 180,E1 -16698.692,E2 -16698.692} C_VEL
LIN {X 0,Y 293.168,Z 226.451,A -85,B 0,C 180,E1 -16699.553,E2 -16699.553} C_VEL
LIN {X 0,Y 291.37,Z 221.505,A -85,B 0,C 180,E1 -16701.03,E2 -16701.03} C_VEL
LIN {X 0,Y 291.339,Z 221.496,A -85,B 0,C 180,E1 -16704.624,E2 -16704.624} C_VEL
LIN {X 0,Y 291.345,Z 221.483,A -85,B 0,C 180,E1 -16707.948,E2 -16707.948} C_VEL
LIN {X 0,Y 291.348,Z 221.508,A -85,B 0,C 180,E1 -16711.155,E2 -16711.155} C_VEL
LIN {X 0,Y 291.387,Z 221.475,A -85,B 0,C 180,E1 -16714.27,E2 -16714.27} C_VEL
LIN {X 0,Y 291.388,Z 221.501,A -85,B 0,C 180,E1 -16717.301,E2 -16717.301} C_VEL
LIN {X 0,Y 291.477,Z 221.455,A -85,B 0,C 180,E1 -16720.272,E2 -16720.272} C_VEL
LIN {X 0,Y 291.513,Z 221.482,A -85,B 0,C 180,E1 -16724.634,E2 -16724.634} C_VEL
LIN {X 0,Y 291.509,Z 221.448,A -85,B 0,C 180,E1 -16728.88,E2 -16728.88} C_VEL
LIN {X 0,Y 291.678,Z 221.464,A -85,B 0,C 180,E1 -16731.688,E2 -16731.688} C_VEL
LIN {X 0,Y 291.601,Z 221.445,A -85,B 0,C 180,E1 -16734.468,E2 -16734.468} C_VEL
LIN {X 0,Y 291.862,Z 221.42,A -85,B 0,C 180,E1 -16738.621,E2 -16738.621} C_VEL
LIN {X 0,Y 291.862,Z 221.441,A -85,B 0,C 180,E1 -16741.381,E2 -16741.381} C_VEL
LIN {X 0,Y 291.707,Z 221.454,A -85,B 0,C 180,E1 -16746.92,E2 -16746.92} C_VEL
LIN {X 0,Y 291.548,Z 221.47,A -85,B 0,C 180,E1 -16749.715,E2 -16749.715} C_VEL
LIN {X 0,Y 291.494,Z 221.478,A -85,B 0,C 180,E1 -16753.952,E2 -16753.952} C_VEL
LIN {X 0,Y 291.461,Z 221.48,A -85,B 0,C 180,E1 -16756.82,E2 -16756.82} C_VEL
LIN {X 0,Y 291.427,Z 221.471,A -85,B 0,C 180,E1 -16759.877,E2 -16759.877} C_VEL
LIN {X 0,Y 291.375,Z 221.488,A -85,B 0,C 180,E1 -16764.208,E2 -16764.208} C_VEL
LIN {X 0,Y 291.398,Z 221.481,A -85,B 0,C 180,E1 -16767.275,E2 -16767.275} C_VEL
LIN {X 0,Y 291.316,Z 221.506,A -85,B 0,C 180,E1 -16770.44,E2 -16770.44} C_VEL
LIN {X 0,Y 291.324,Z 221.487,A -85,B 0,C 180,E1 -16773.702,E2 -16773.702} C_VEL
LIN {X 0,Y 291.353,Z 221.501,A -85,B 0,C 180,E1 -16777.256,E2 -16777.256} C_VEL
LIN {X 0,Y 291.315,Z 221.496,A -85,B 0,C 180,E1 -16780.647,E2 -16780.647} C_VEL
LIN {X 0,Y 291.275,Z 221.496,A -85,B 0,C 180,E1 -16784.406,E2 -16784.406} C_VEL
LIN {X 0,Y 291.312,Z 221.51,A -85,B 0,C 180,E1 -16788.409,E2 -16788.409} C_VEL
LIN {X 0,Y 291.327,Z 221.493,A -85,B 0,C 180,E1 -16791.16,E2 -16791.16} C_VEL
LIN {X 0,Y 291.35,Z 221.492,A -85,B 0,C 180,E1 -16794.63,E2 -16794.63} C_VEL
LIN {X 0,Y 291.357,Z 221.508,A -85,B 0,C 180,E1 -16797.954,E2 -16797.954} C_VEL
LIN {X 0,Y 291.337,Z 221.5,A -85,B 0,C 180,E1 -16801.159,E2 -16801.159} C_VEL
LIN {X 0,Y 291.355,Z 221.493,A -85,B 0,C 180,E1 -16804.271,E2 -16804.271} C_VEL
LIN {X 0,Y 291.379,Z 221.622,A -85,B 0,C 180,E1 -16807.475,E2 -16807.475} C_VEL
LIN {X 0,Y 292.35,Z 224.324,A -85,B 0,C 180,E1 -16807.766,E2 -16807.766} C_VEL
LIN {X 0,Y 294.5,Z 226.769,A -85,B 0,C 180,E1 -16808.274,E2 -16808.274} C_VEL
LIN {X 0,Y 296.682,Z 230.2,A -85,B 0,C 180,E1 -16808.816,E2 -16808.816} C_VEL
LIN {X 0,Y 298.202,Z 232.292,A -85,B 0,C 180,E1 -16809.176,E2 -16809.176} C_VEL
LIN {X 0,Y 306.207,Z 244.053,A -85,B 0,C 180,E1 -16811.009,E2 -16811.009} C_VEL
LIN {X 0,Y 314.88,Z 257.507,A -85,B 0,C 180,E1 -16812.873,E2 -16812.873} C_VEL
LIN {X 0,Y 324.583,Z 274.123,A -85,B 0,C 180,E1 -16814.846,E2 -16814.846} C_VEL
LIN {X 0,Y 329.598,Z 284.583,A -85,B 0,C 180,E1 -16815.86,E2 -16815.86} C_VEL
LIN {X 0,Y 323.31,Z 420.139,A -85,B 0,C 180,E1 -16818.924,E2 -16818.924} C_VEL
LIN {X 0,Y 321.752,Z 437.556,A -85,B 0,C 180,E1 -16819.561,E2 -16819.561} C_VEL
LIN {X 0,Y 319.728,Z 454.244,A -85,B 0,C 180,E1 -16820.435,E2 -16820.435} C_VEL
LIN {X 0,Y 317.417,Z 469.589,A -85,B 0,C 180,E1 -16821.488,E2 -16821.488} C_VEL
LIN {X 0,Y 314.709,Z 484.725,A -85,B 0,C 180,E1 -16822.787,E2 -16822.787} C_VEL
LIN {X 0,Y 311.668,Z 499.47,A -85,B 0,C 180,E1 -16824.342,E2 -16824.342} C_VEL
LIN {X 0,Y 308.562,Z 513.075,A -85,B 0,C 180,E1 -16826.085,E2 -16826.085} C_VEL
LIN {X 0,Y 305.357,Z 525.646,A -85,B 0,C 180,E1 -16828.025,E2 -16828.025} C_VEL
LIN {X 0,Y 302.212,Z 537.79,A -85,B 0,C 180,E1 -16830.275,E2 -16830.275} C_VEL
LIN {X 0,Y 299.23,Z 548.729,A -85,B 0,C 180,E1 -16832.696,E2 -16832.696} C_VEL
LIN {X 0,Y 296.683,Z 558.186,A -85,B 0,C 180,E1 -16835.193,E2 -16835.193} C_VEL
LIN {X 0,Y 294.417,Z 566.645,A -85,B 0,C 180,E1 -16837.892,E2 -16837.892} C_VEL
LIN {X 0,Y 292.876,Z 572.942,A -85,B 0,C 180,E1 -16840.304,E2 -16840.304} C_VEL
LIN {X 0,Y 291.417,Z 579.315,A -85,B 0,C 180,E1 -16843.247,E2 -16843.247} C_VEL
LIN {X 0,Y 290.438,Z 584.223,A -85,B 0,C 180,E1 -16846.16,E2 -16846.16} C_VEL
LIN {X 0,Y 289.762,Z 587.821,A -85,B 0,C 180,E1 -16848.926,E2 -16848.926} C_VEL
LIN {X 0,Y 289.172,Z 591.002,A -85,B 0,C 180,E1 -16852.548,E2 -16852.548} C_VEL
LIN {X 0,Y 289.036,Z 592.507,A -85,B 0,C 180,E1 -16855.958,E2 -16855.958} C_VEL
LIN {X 0,Y 289.129,Z 592.585,A -85,B 0,C 180,E1 -16859.09,E2 -16859.09} C_VEL
LIN {X 0,Y 289.334,Z 591.431,A -85,B 0,C 180,E1 -16862.305,E2 -16862.305} C_VEL
LIN {X 0,Y 289.88,Z 588.964,A -85,B 0,C 180,E1 -16865.585,E2 -16865.585} C_VEL
LIN {X 0,Y 290.622,Z 586.154,A -85,B 0,C 180,E1 -16868.075,E2 -16868.075} C_VEL
LIN {X 0,Y 291.84,Z 581.486,A -85,B 0,C 180,E1 -16871.183,E2 -16871.183} C_VEL
LIN {X 0,Y 293.378,Z 575.972,A -85,B 0,C 180,E1 -16874.055,E2 -16874.055} C_VEL
LIN {X 0,Y 295.344,Z 569.373,A -85,B 0,C 180,E1 -16876.795,E2 -16876.795} C_VEL
LIN {X 0,Y 297.945,Z 561.503,A -85,B 0,C 180,E1 -16879.483,E2 -16879.483} C_VEL
LIN {X 0,Y 300.848,Z 552.543,A -85,B 0,C 180,E1 -16882.041,E2 -16882.041} C_VEL
LIN {X 0,Y 304.106,Z 542.41,A -85,B 0,C 180,E1 -16884.439,E2 -16884.439} C_VEL
LIN {X 0,Y 306.379,Z 535.091,A -85,B 0,C 180,E1 -16885.935,E2 -16885.935} C_VEL
LIN {X 0,Y 307.025,Z 531.15,A -85,B 0,C 180,E1 -16886.752,E2 -16886.752} C_VEL
LIN {X 0,Y 306.174,Z 519.578,A -85,B 0,C 180,E1 -16889.289,E2 -16889.289} C_VEL
LIN {X 0,Y 306.606,Z 515.26,A -85,B 0,C 180,E1 -16890.035,E2 -16890.035} C_VEL
LIN {X 0,Y 306.983,Z 513.732,A -85,B 0,C 180,E1 -16890.255,E2 -16890.255} C_VEL
LIN {X 0,Y 310.587,Z 500.61,A -85,B 0,C 180,E1 -16891.948,E2 -16891.948} C_VEL
LIN {X 0,Y 314.163,Z 486.053,A -85,B 0,C 180,E1 -16893.488,E2 -16893.488} C_VEL
LIN {X 0,Y 317.23,Z 471.863,A -85,B 0,C 180,E1 -16894.714,E2 -16894.714} C_VEL
LIN {X 0,Y 319.954,Z 456.811,A -85,B 0,C 180,E1 -16895.77,E2 -16895.77} C_VEL
LIN {X 0,Y 322.217,Z 441.252,A -85,B 0,C 180,E1 -16896.606,E2 -16896.606} C_VEL
LIN {X 0,Y 323.92,Z 425.705,A -85,B 0,C 180,E1 -16897.217,E2 -16897.217} C_VEL
LIN {X 0,Y 325.354,Z 403.769,A -85,B 0,C 180,E1 -16897.8,E2 -16897.8} C_VEL
LIN {X 0,Y 331.692,Z 291.163,A -85,B 0,C 180,E1 -16900.374,E2 -16900.374} C_VEL
LIN {X 0,Y 325.206,Z 278.342,A -85,B 0,C 180,E1 -16902.124,E2 -16902.124} C_VEL
LIN {X 0,Y 317.514,Z 266.008,A -85,B 0,C 180,E1 -16904.314,E2 -16904.314} C_VEL
LIN {X 0,Y 311.59,Z 257.14,A -85,B 0,C 180,E1 -16906.168,E2 -16906.168} C_VEL
LIN {X 0,Y 305.109,Z 248.286,A -85,B 0,C 180,E1 -16908.396,E2 -16908.396} C_VEL
LIN {X 0,Y 302.253,Z 244.468,A -85,B 0,C 180,E1 -16909.477,E2 -16909.477} C_VEL
LIN {X 0,Y 298.792,Z 240.32,A -85,B 0,C 180,E1 -16910.842,E2 -16910.842} C_VEL
LIN {X 0,Y 297.665,Z 238.682,A -85,B 0,C 180,E1 -16911.325,E2 -16911.325} C_VEL
LIN {X 0,Y 295.137,Z 235.841,A -85,B 0,C 180,E1 -16912.431,E2 -16912.431} C_VEL
LIN {X 0,Y 293.909,Z 233.677,A -85,B 0,C 180,E1 -16913.046,E2 -16913.046} C_VEL
LIN {X 0,Y 291.082,Z 231.338,A -85,B 0,C 180,E1 -16914.37,E2 -16914.37} C_VEL
LIN {X 0,Y 289.49,Z 228.434,A -85,B 0,C 180,E1 -16915.264,E2 -16915.264} C_VEL
LIN {X 0,Y 286.735,Z 226.551,A -85,B 0,C 180,E1 -16916.75,E2 -16916.75} C_VEL
LIN {X 0,Y 285.175,Z 223.929,A -85,B 0,C 180,E1 -16917.792,E2 -16917.792} C_VEL
LIN {X 0,Y 284.8,Z 222.32,A -85,B 0,C 180,E1 -16918.143,E2 -16918.143} C_VEL
LIN {X 0,Y 284.857,Z 222.309,A -85,B 0,C 180,E1 -16921.413,E2 -16921.413} C_VEL
LIN {X 0,Y 284.658,Z 222.333,A -85,B 0,C 180,E1 -16927.09,E2 -16927.09} C_VEL
LIN {X 0,Y 284.518,Z 222.35,A -85,B 0,C 180,E1 -16929.956,E2 -16929.956} C_VEL
LIN {X 0,Y 284.467,Z 222.362,A -85,B 0,C 180,E1 -16934.303,E2 -16934.303} C_VEL
LIN {X 0,Y 284.336,Z 222.372,A -85,B 0,C 180,E1 -16938.742,E2 -16938.742} C_VEL
LIN {X 0,Y 284.337,Z 222.379,A -85,B 0,C 180,E1 -16943.295,E2 -16943.295} C_VEL
LIN {X 0,Y 284.399,Z 222.365,A -85,B 0,C 180,E1 -16947.171,E2 -16947.171} C_VEL
LIN {X 0,Y 284.357,Z 222.547,A -85,B 0,C 180,E1 -16948.107,E2 -16948.107} C_VEL
LIN {X 0,Y 284.591,Z 223.591,A -85,B 0,C 180,E1 -16948.484,E2 -16948.484} C_VEL
LIN {X 0,Y 285.829,Z 225.935,A -85,B 0,C 180,E1 -16949.355,E2 -16949.355} C_VEL
LIN {X 0,Y 288.846,Z 228.586,A -85,B 0,C 180,E1 -16951.082,E2 -16951.082} C_VEL
LIN {X 0,Y 292.015,Z 232.69,A -85,B 0,C 180,E1 -16952.745,E2 -16952.745} C_VEL
LIN {X 0,Y 293.48,Z 234.588,A -85,B 0,C 180,E1 -16953.467,E2 -16953.467} C_VEL
LIN {X 0,Y 296.165,Z 237.87,A -85,B 0,C 180,E1 -16954.716,E2 -16954.716} C_VEL
LIN {X 0,Y 298.524,Z 241.183,A -85,B 0,C 180,E1 -16955.742,E2 -16955.742} C_VEL
LIN {X 0,Y 301.717,Z 245.596,A -85,B 0,C 180,E1 -16957.038,E2 -16957.038} C_VEL
LIN {X 0,Y 306.108,Z 252.002,A -85,B 0,C 180,E1 -16958.711,E2 -16958.711} C_VEL
LIN {X 0,Y 311.451,Z 260.215,A -85,B 0,C 180,E1 -16960.561,E2 -16960.561} C_VEL
LIN {X 0,Y 317.982,Z 271.167,A -85,B 0,C 180,E1 -16962.633,E2 -16962.633} C_VEL
LIN {X 0,Y 324.236,Z 282.689,A -85,B 0,C 180,E1 -16964.463,E2 -16964.463} C_VEL
LIN {X 0,Y 330.518,Z 295.833,A -85,B 0,C 180,E1 -16966.194,E2 -16966.194} C_VEL
LIN {X 0,Y 331.427,Z 298.209,A -85,B 0,C 180,E1 -16966.45,E2 -16966.45} C_VEL
LIN {X 0,Y 323.785,Z 433.995,A -85,B 0,C 180,E1 -16969.586,E2 -16969.586} C_VEL
LIN {X 0,Y 321.826,Z 451.632,A -85,B 0,C 180,E1 -16970.204,E2 -16970.204} C_VEL
LIN {X 0,Y 319.251,Z 468.354,A -85,B 0,C 180,E1 -16971.038,E2 -16971.038} C_VEL
LIN {X 0,Y 316.562,Z 482.603,A -85,B 0,C 180,E1 -16971.968,E2 -16971.968} C_VEL
LIN {X 0,Y 313.445,Z 497.069,A -85,B 0,C 180,E1 -16973.144,E2 -16973.144} C_VEL
LIN {X 0,Y 309.699,Z 511.98,A -85,B 0,C 180,E1 -16974.641,E2 -16974.641} C_VEL
LIN {X 0,Y 305.895,Z 525.684,A -85,B 0,C 180,E1 -16976.337,E2 -16976.337} C_VEL
LIN {X 0,Y 302.356,Z 537.455,A -85,B 0,C 180,E1 -16978.073,E2 -16978.073} C_VEL
LIN {X 0,Y 298.327,Z 550.284,A -85,B 0,C 180,E1 -16980.346,E2 -16980.346} C_VEL
LIN {X 0,Y 294.807,Z 561.19,A -85,B 0,C 180,E1 -16982.681,E2 -16982.681} C_VEL
LIN {X 0,Y 291.29,Z 571.778,A -85,B 0,C 180,E1 -16985.403,E2 -16985.403} C_VEL
LIN {X 0,Y 288.617,Z 580.155,A -85,B 0,C 180,E1 -16987.999,E2 -16987.999} C_VEL
LIN {X 0,Y 286.511,Z 587.362,A -85,B 0,C 180,E1 -16990.659,E2 -16990.659} C_VEL
LIN {X 0,Y 284.442,Z 595.106,A -85,B 0,C 180,E1 -16994.226,E2 -16994.226} C_VEL
LIN {X 0,Y 283.12,Z 601.042,A -85,B 0,C 180,E1 -16997.816,E2 -16997.816} C_VEL
LIN {X 0,Y 282.432,Z 605.295,A -85,B 0,C 180,E1 -17001.41,E2 -17001.41} C_VEL
LIN {X 0,Y 282.326,Z 607.781,A -85,B 0,C 180,E1 -17004.696,E2 -17004.696} C_VEL
LIN {X 0,Y 282.327,Z 608.841,A -85,B 0,C 180,E1 -17007.143,E2 -17007.143} C_VEL
LIN {X 0,Y 282.354,Z 609.109,A -85,B 0,C 180,E1 -17009.997,E2 -17009.997} C_VEL
LIN {X 0,Y 282.337,Z 608.44,A -85,B 0,C 180,E1 -17012.85,E2 -17012.85} C_VEL
LIN {X 0,Y 282.33,Z 606.714,A -85,B 0,C 180,E1 -17015.711,E2 -17015.711} C_VEL
LIN {X 0,Y 282.426,Z 604.028,A -85,B 0,C 180,E1 -17018.583,E2 -17018.583} C_VEL
LIN {X 0,Y 283.078,Z 599.108,A -85,B 0,C 180,E1 -17022.179,E2 -17022.179} C_VEL
LIN {X 0,Y 284.141,Z 593.389,A -85,B 0,C 180,E1 -17025.286,E2 -17025.286} C_VEL
LIN {X 0,Y 285.356,Z 587.426,A -85,B 0,C 180,E1 -17027.926,E2 -17027.926} C_VEL
LIN {X 0,Y 287.307,Z 579.61,A -85,B 0,C 180,E1 -17030.77,E2 -17030.77} C_VEL
LIN {X 0,Y 289.754,Z 570.194,A -85,B 0,C 180,E1 -17033.587,E2 -17033.587} C_VEL
LIN {X 0,Y 292.445,Z 560.489,A -85,B 0,C 180,E1 -17036.009,E2 -17036.009} C_VEL
LIN {X 0,Y 295.538,Z 549.146,A -85,B 0,C 180,E1 -17038.394,E2 -17038.394} C_VEL
LIN {X 0,Y 298.896,Z 536.781,A -85,B 0,C 180,E1 -17040.557,E2 -17040.557} C_VEL
LIN {X 0,Y 302.331,Z 523.249,A -85,B 0,C 180,E1 -17042.513,E2 -17042.513} C_VEL
LIN {X 0,Y 305.586,Z 509.452,A -85,B 0,C 180,E1 -17044.159,E2 -17044.159} C_VEL
LIN {X 0,Y 308.547,Z 495.804,A -85,B 0,C 180,E1 -17045.504,E2 -17045.504} C_VEL
LIN {X 0,Y 311.367,Z 480.596,A -85,B 0,C 180,E1 -17046.731,E2 -17046.731} C_VEL
LIN {X 0,Y 313.974,Z 463.686,A -85,B 0,C 180,E1 -17047.784,E2 -17047.784} C_VEL
LIN {X 0,Y 315.994,Z 447.597,A -85,B 0,C 180,E1 -17048.511,E2 -17048.511} C_VEL
LIN {X 0,Y 317.417,Z 430.65,A -85,B 0,C 180,E1 -17049.052,E2 -17049.052} C_VEL
LIN {X 0,Y 323.817,Z 294.498,A -85,B 0,C 180,E1 -17052.165,E2 -17052.165} C_VEL
LIN {X 0,Y 314.385,Z 274.985,A -85,B 0,C 180,E1 -17054.164,E2 -17054.164} C_VEL
LIN {X 0,Y 304.228,Z 256.183,A -85,B 0,C 180,E1 -17056.435,E2 -17056.435} C_VEL
LIN {X 0,Y 294.269,Z 239.626,A -85,B 0,C 180,E1 -17058.82,E2 -17058.82} C_VEL
LIN {X 0,Y 285.743,Z 226.292,A -85,B 0,C 180,E1 -17061.045,E2 -17061.045} C_VEL
LIN {X 0,Y 284.314,Z 222.369,A -85,B 0,C 180,E1 -17062.319,E2 -17062.319} C_VEL
LIN {X 0,Y 284.286,Z 222.385,A -85,B 0,C 180,E1 -17065.348,E2 -17065.348} C_VEL
LIN {X 0,Y 284.268,Z 222.366,A -85,B 0,C 180,E1 -17068.723,E2 -17068.723} C_VEL
LIN {X 0,Y 284.366,Z 222.352,A -85,B 0,C 180,E1 -17072.827,E2 -17072.827} C_VEL
LIN {X 0,Y 284.354,Z 222.38,A -85,B 0,C 180,E1 -17076.707,E2 -17076.707} C_VEL
LIN {X 0,Y 284.405,Z 222.336,A -85,B 0,C 180,E1 -17079.873,E2 -17079.873} C_VEL
LIN {X 0,Y 284.451,Z 222.364,A -85,B 0,C 180,E1 -17084.469,E2 -17084.469} C_VEL
LIN {X 0,Y 284.461,Z 222.322,A -85,B 0,C 180,E1 -17088.601,E2 -17088.601} C_VEL
LIN {X 0,Y 284.629,Z 222.343,A -85,B 0,C 180,E1 -17091.481,E2 -17091.481} C_VEL
LIN {X 0,Y 284.571,Z 222.322,A -85,B 0,C 180,E1 -17094.331,E2 -17094.331} C_VEL
LIN {X 0,Y 284.828,Z 222.294,A -85,B 0,C 180,E1 -17098.587,E2 -17098.587} C_VEL
LIN {X 0,Y 284.828,Z 222.317,A -85,B 0,C 180,E1 -17101.415,E2 -17101.415} C_VEL
LIN {X 0,Y 284.658,Z 222.334,A -85,B 0,C 180,E1 -17107.092,E2 -17107.092} C_VEL
LIN {X 0,Y 284.492,Z 222.343,A -85,B 0,C 180,E1 -17109.959,E2 -17109.959} C_VEL
LIN {X 0,Y 284.451,Z 222.358,A -85,B 0,C 180,E1 -17114.305,E2 -17114.305} C_VEL
LIN {X 0,Y 284.4,Z 222.355,A -85,B 0,C 180,E1 -17117.251,E2 -17117.251} C_VEL
LIN {X 0,Y 284.355,Z 222.356,A -85,B 0,C 180,E1 -17120.245,E2 -17120.245} C_VEL
LIN {X 0,Y 284.345,Z 222.369,A -85,B 0,C 180,E1 -17123.877,E2 -17123.877} C_VEL
LIN {X 0,Y 284.373,Z 222.353,A -85,B 0,C 180,E1 -17127.176,E2 -17127.176} C_VEL
LIN {X 0,Y 284.274,Z 222.374,A -85,B 0,C 180,E1 -17131.278,E2 -17131.278} C_VEL
LIN {X 0,Y 284.322,Z 222.379,A -85,B 0,C 180,E1 -17135.351,E2 -17135.351} C_VEL
LIN {X 0,Y 284.29,Z 222.366,A -85,B 0,C 180,E1 -17138.174,E2 -17138.174} C_VEL
LIN {X 0,Y 284.253,Z 222.391,A -85,B 0,C 180,E1 -17142.128,E2 -17142.128} C_VEL
LIN {X 0,Y 284.24,Z 222.375,A -85,B 0,C 180,E1 -17146.193,E2 -17146.193} C_VEL
LIN {X 0,Y 284.294,Z 222.368,A -85,B 0,C 180,E1 -17150.028,E2 -17150.028} C_VEL
LIN {X 0,Y 284.317,Z 222.38,A -85,B 0,C 180,E1 -17153.618,E2 -17153.618} C_VEL
LIN {X 0,Y 284.297,Z 222.382,A -85,B 0,C 180,E1 -17157.195,E2 -17157.195} C_VEL
LIN {X 0,Y 284.329,Z 222.366,A -85,B 0,C 180,E1 -17160.378,E2 -17160.378} C_VEL
LIN {X 0,Y 284.3,Z 222.373,A -85,B 0,C 180,E1 -17163.584,E2 -17163.584} C_VEL
LIN {X 0,Y 284.316,Z 222.383,A -85,B 0,C 180,E1 -17166.044,E2 -17166.044} C_VEL
LIN {X 0,Y 285.346,Z 225.237,A -85,B 0,C 180,E1 -17166.373,E2 -17166.373} C_VEL
LIN {X 0,Y 287.612,Z 227.861,A -85,B 0,C 180,E1 -17166.945,E2 -17166.945} C_VEL
LIN {X 0,Y 289.682,Z 231.089,A -85,B 0,C 180,E1 -17167.485,E2 -17167.485} C_VEL
LIN {X 0,Y 291.017,Z 232.834,A -85,B 0,C 180,E1 -17167.814,E2 -17167.814} C_VEL
LIN {X 0,Y 299.454,Z 245.007,A -85,B 0,C 180,E1 -17169.849,E2 -17169.849} C_VEL
LIN {X 0,Y 309.407,Z 260.43,A -85,B 0,C 180,E1 -17172.081,E2 -17172.081} C_VEL
LIN {X 0,Y 319.549,Z 277.758,A -85,B 0,C 180,E1 -17174.217,E2 -17174.217} C_VEL
LIN {X 0,Y 323.852,Z 286.416,A -85,B 0,C 180,E1 -17175.105,E2 -17175.105} C_VEL
LIN {X 0,Y 317.528,Z 420.307,A -85,B 0,C 180,E1 -17178.19,E2 -17178.19} C_VEL
LIN {X 0,Y 315.905,Z 437.947,A -85,B 0,C 180,E1 -17178.843,E2 -17178.843} C_VEL
LIN {X 0,Y 313.919,Z 453.861,A -85,B 0,C 180,E1 -17179.686,E2 -17179.686} C_VEL
LIN {X 0,Y 311.545,Z 469.342,A -85,B 0,C 180,E1 -17180.754,E2 -17180.754} C_VEL
LIN {X 0,Y 308.572,Z 485.387,A -85,B 0,C 180,E1 -17182.149,E2 -17182.149} C_VEL
LIN {X 0,Y 305.454,Z 499.895,A -85,B 0,C 180,E1 -17183.707,E2 -17183.707} C_VEL
LIN {X 0,Y 302.306,Z 513.274,A -85,B 0,C 180,E1 -17185.453,E2 -17185.453} C_VEL
LIN {X 0,Y 299.167,Z 525.157,A -85,B 0,C 180,E1 -17187.31,E2 -17187.31} C_VEL
LIN {X 0,Y 295.792,Z 537.723,A -85,B 0,C 180,E1 -17189.663,E2 -17189.663} C_VEL
LIN {X 0,Y 292.758,Z 548.451,A -85,B 0,C 180,E1 -17192.067,E2 -17192.067} C_VEL
LIN {X 0,Y 289.963,Z 558.362,A -85,B 0,C 180,E1 -17194.729,E2 -17194.729} C_VEL
LIN {X 0,Y 287.403,Z 567.534,A -85,B 0,C 180,E1 -17197.732,E2 -17197.732} C_VEL
LIN {X 0,Y 285.512,Z 574.958,A -85,B 0,C 180,E1 -17200.754,E2 -17200.754} C_VEL
LIN {X 0,Y 284.17,Z 580.601,A -85,B 0,C 180,E1 -17203.592,E2 -17203.592} C_VEL
LIN {X 0,Y 283.224,Z 585.347,A -85,B 0,C 180,E1 -17206.584,E2 -17206.584} C_VEL
LIN {X 0,Y 282.627,Z 588.341,A -85,B 0,C 180,E1 -17209.1,E2 -17209.1} C_VEL
LIN {X 0,Y 282.167,Z 590.858,A -85,B 0,C 180,E1 -17211.941,E2 -17211.941} C_VEL
LIN {X 0,Y 281.95,Z 592.424,A -85,B 0,C 180,E1 -17215.074,E2 -17215.074} C_VEL
LIN {X 0,Y 281.99,Z 592.883,A -85,B 0,C 180,E1 -17218.267,E2 -17218.267} C_VEL
LIN {X 0,Y 282.178,Z 592.151,A -85,B 0,C 180,E1 -17221.538,E2 -17221.538} C_VEL
LIN {X 0,Y 282.648,Z 590.04,A -85,B 0,C 180,E1 -17224.885,E2 -17224.885} C_VEL
LIN {X 0,Y 283.611,Z 586.527,A -85,B 0,C 180,E1 -17228.283,E2 -17228.283} C_VEL
LIN {X 0,Y 284.998,Z 581.452,A -85,B 0,C 180,E1 -17231.747,E2 -17231.747} C_VEL
LIN {X 0,Y 286.694,Z 575.861,A -85,B 0,C 180,E1 -17234.69,E2 -17234.69} C_VEL
LIN {X 0,Y 289.149,Z 568.311,A -85,B 0,C 180,E1 -17237.847,E2 -17237.847} C_VEL
LIN {X 0,Y 292.32,Z 559.097,A -85,B 0,C 180,E1 -17240.914,E2 -17240.914} C_VEL
LIN {X 0,Y 295.539,Z 549.523,A -85,B 0,C 180,E1 -17243.522,E2 -17243.522} C_VEL
LIN {X 0,Y 299.102,Z 538.952,A -85,B 0,C 180,E1 -17245.923,E2 -17245.923} C_VEL
LIN {X 0,Y 302.915,Z 527.231,A -85,B 0,C 180,E1 -17248.142,E2 -17248.142} C_VEL
LIN {X 0,Y 306.76,Z 514.505,A -85,B 0,C 180,E1 -17250.15,E2 -17250.15} C_VEL
LIN {X 0,Y 306.983,Z 513.732,A -85,B 0,C 180,E1 -17250.255,E2 -17250.255} C_VEL
LIN {X 0,Y 307.749,Z 509.232,A -85,B 0,C 180,E1 -17250.946,E2 -17250.946} C_VEL
LIN {X 0,Y 307.201,Z 494.503,A -85,B 0,C 180,E1 -17253.429,E2 -17253.429} C_VEL
LIN {X 0,Y 307.947,Z 489.581,A -85,B 0,C 180,E1 -17254.016,E2 -17254.016} C_VEL
LIN {X 0,Y 311.278,Z 475.224,A -85,B 0,C 180,E1 -17255.337,E2 -17255.337} C_VEL
LIN {X 0,Y 314.273,Z 459.677,A -85,B 0,C 180,E1 -17256.475,E2 -17256.475} C_VEL
LIN {X 0,Y 316.727,Z 444.007,A -85,B 0,C 180,E1 -17257.363,E2 -17257.363} C_VEL
LIN {X 0,Y 318.717,Z 427.36,A -85,B 0,C 180,E1 -17258.053,E2 -17258.053} C_VEL
LIN {X 0,Y 320.088,Z 409.057,A -85,B 0,C 180,E1 -17258.567,E2 -17258.567} C_VEL
LIN {X 0,Y 326.802,Z 293.817,A -85,B 0,C 180,E1 -17261.246,E2 -17261.246} C_VEL
LIN {X 0,Y 321.198,Z 282.872,A -85,B 0,C 180,E1 -17262.821,E2 -17262.821} C_VEL
LIN {X 0,Y 314.811,Z 272.388,A -85,B 0,C 180,E1 -17264.71,E2 -17264.71} C_VEL
LIN {X 0,Y 308.678,Z 262.986,A -85,B 0,C 180,E1 -17266.697,E2 -17266.697} C_VEL
LIN {X 0,Y 302.327,Z 254.166,A -85,B 0,C 180,E1 -17268.972,E2 -17268.972} C_VEL
LIN {X 0,Y 298.938,Z 249.682,A -85,B 0,C 180,E1 -17270.302,E2 -17270.302} C_VEL
LIN {X 0,Y 295.964,Z 245.714,A -85,B 0,C 180,E1 -17271.555,E2 -17271.555} C_VEL
LIN {X 0,Y 292.599,Z 241.525,A -85,B 0,C 180,E1 -17273.102,E2 -17273.102} C_VEL
LIN {X 0,Y 291.606,Z 240.055,A -85,B 0,C 180,E1 -17273.599,E2 -17273.599} C_VEL
LIN {X 0,Y 288.781,Z 237.333,A -85,B 0,C 180,E1 -17274.994,E2 -17274.994} C_VEL
LIN {X 0,Y 287.417,Z 234.9,A -85,B 0,C 180,E1 -17275.792,E2 -17275.792} C_VEL
LIN {X 0,Y 284.992,Z 233.076,A -85,B 0,C 180,E1 -17277.172,E2 -17277.172} C_VEL
LIN {X 0,Y 283.214,Z 230.106,A -85,B 0,C 180,E1 -17278.4,E2 -17278.4} C_VEL
LIN {X 0,Y 282.754,Z 229.09,A -85,B 0,C 180,E1 -17278.753,E2 -17278.753} C_VEL
LIN {X 0,Y 279.737,Z 227.219,A -85,B 0,C 180,E1 -17280.899,E2 -17280.899} C_VEL
LIN {X 0,Y 278.091,Z 224.766,A -85,B 0,C 180,E1 -17282.443,E2 -17282.443} C_VEL
LIN {X 0,Y 277.641,Z 223.215,A -85,B 0,C 180,E1 -17283.083,E2 -17283.083} C_VEL
LIN {X 0,Y 277.616,Z 223.209,A -85,B 0,C 180,E1 -17287.271,E2 -17287.271} C_VEL
LIN {X 0,Y 277.462,Z 223.228,A -85,B 0,C 180,E1 -17290.212,E2 -17290.212} C_VEL
LIN {X 0,Y 277.413,Z 223.243,A -85,B 0,C 180,E1 -17294.675,E2 -17294.675} C_VEL
LIN {X 0,Y 277.289,Z 223.25,A -85,B 0,C 180,E1 -17299.237,E2 -17299.237} C_VEL
LIN {X 0,Y 277.327,Z 223.407,A -85,B 0,C 180,E1 -17303.375,E2 -17303.375} C_VEL
LIN {X 0,Y 277.992,Z 225.571,A -85,B 0,C 180,E1 -17304.198,E2 -17304.198} C_VEL
LIN {X 0,Y 279.836,Z 227.856,A -85,B 0,C 180,E1 -17305.872,E2 -17305.872} C_VEL
LIN {X 0,Y 282.546,Z 229.436,A -85,B 0,C 180,E1 -17307.783,E2 -17307.783} C_VEL
LIN {X 0,Y 283.991,Z 232.337,A -85,B 0,C 180,E1 -17308.853,E2 -17308.853} C_VEL
LIN {X 0,Y 286.498,Z 234.6,A -85,B 0,C 180,E1 -17310.362,E2 -17310.362} C_VEL
LIN {X 0,Y 288.309,Z 237.104,A -85,B 0,C 180,E1 -17311.408,E2 -17311.408} C_VEL
LIN {X 0,Y 291.247,Z 240.729,A -85,B 0,C 180,E1 -17312.924,E2 -17312.924} C_VEL
LIN {X 0,Y 293.932,Z 244.169,A -85,B 0,C 180,E1 -17314.22,E2 -17314.22} C_VEL
LIN {X 0,Y 296.615,Z 247.888,A -85,B 0,C 180,E1 -17315.433,E2 -17315.433} C_VEL
LIN {X 0,Y 302.535,Z 256.616,A -85,B 0,C 180,E1 -17317.846,E2 -17317.846} C_VEL
LIN {X 0,Y 307.952,Z 264.972,A -85,B 0,C 180,E1 -17319.823,E2 -17319.823} C_VEL
LIN {X 0,Y 315.372,Z 277.795,A -85,B 0,C 180,E1 -17322.277,E2 -17322.277} C_VEL
LIN {X 0,Y 321.756,Z 290.131,A -85,B 0,C 180,E1 -17324.207,E2 -17324.207} C_VEL
LIN {X 0,Y 326.533,Z 300.545,A -85,B 0,C 180,E1 -17325.571,E2 -17325.571} C_VEL
LIN {X 0,Y 318.743,Z 433.709,A -85,B 0,C 180,E1 -17328.693,E2 -17328.693} C_VEL
LIN {X 0,Y 316.785,Z 450.907,A -85,B 0,C 180,E1 -17329.298,E2 -17329.298} C_VEL
LIN {X 0,Y 314.254,Z 466.962,A -85,B 0,C 180,E1 -17330.089,E2 -17330.089} C_VEL
LIN {X 0,Y 311.039,Z 483.435,A -85,B 0,C 180,E1 -17331.167,E2 -17331.167} C_VEL
LIN {X 0,Y 307.446,Z 499.231,A -85,B 0,C 180,E1 -17332.507,E2 -17332.507} C_VEL
LIN {X 0,Y 303.95,Z 512.454,A -85,B 0,C 180,E1 -17333.869,E2 -17333.869} C_VEL
LIN {X 0,Y 299.643,Z 527.175,A -85,B 0,C 180,E1 -17335.74,E2 -17335.74} C_VEL
LIN {X 0,Y 295.701,Z 539.639,A -85,B 0,C 180,E1 -17337.67,E2 -17337.67} C_VEL
LIN {X 0,Y 291.654,Z 551.789,A -85,B 0,C 180,E1 -17339.926,E2 -17339.926} C_VEL
LIN {X 0,Y 287.938,Z 562.72,A -85,B 0,C 180,E1 -17342.368,E2 -17342.368} C_VEL
LIN {X 0,Y 284.348,Z 573.057,A -85,B 0,C 180,E1 -17345.152,E2 -17345.152} C_VEL
LIN {X 0,Y 281.455,Z 581.708,A -85,B 0,C 180,E1 -17348,E2 -17348} C_VEL
LIN {X 0,Y 279.198,Z 588.973,A -85,B 0,C 180,E1 -17350.896,E2 -17350.896} C_VEL
LIN {X 0,Y 277.5,Z 595.033,A -85,B 0,C 180,E1 -17353.821,E2 -17353.821} C_VEL
LIN {X 0,Y 276.13,Z 600.931,A -85,B 0,C 180,E1 -17357.503,E2 -17357.503} C_VEL
LIN {X 0,Y 275.363,Z 605.151,A -85,B 0,C 180,E1 -17361.188,E2 -17361.188} C_VEL
LIN {X 0,Y 275.226,Z 607.742,A -85,B 0,C 180,E1 -17364.789,E2 -17364.789} C_VEL
LIN {X 0,Y 275.235,Z 608.656,A -85,B 0,C 180,E1 -17367.069,E2 -17367.069} C_VEL
LIN {X 0,Y 275.276,Z 608.896,A -85,B 0,C 180,E1 -17369.996,E2 -17369.996} C_VEL
LIN {X 0,Y 275.245,Z 608.212,A -85,B 0,C 180,E1 -17372.924,E2 -17372.924} C_VEL
LIN {X 0,Y 275.225,Z 606.454,A -85,B 0,C 180,E1 -17375.859,E2 -17375.859} C_VEL
LIN {X 0,Y 275.357,Z 603.75,A -85,B 0,C 180,E1 -17378.805,E2 -17378.805} C_VEL
LIN {X 0,Y 276.049,Z 598.796,A -85,B 0,C 180,E1 -17382.494,E2 -17382.494} C_VEL
LIN {X 0,Y 277.084,Z 593.477,A -85,B 0,C 180,E1 -17385.458,E2 -17385.458} C_VEL
LIN {X 0,Y 278.495,Z 587.035,A -85,B 0,C 180,E1 -17388.383,E2 -17388.383} C_VEL
LIN {X 0,Y 280.524,Z 579.195,A -85,B 0,C 180,E1 -17391.297,E2 -17391.297} C_VEL
LIN {X 0,Y 283.14,Z 569.732,A -85,B 0,C 180,E1 -17394.172,E2 -17394.172} C_VEL
LIN {X 0,Y 285.97,Z 559.973,A -85,B 0,C 180,E1 -17396.643,E2 -17396.643} C_VEL
LIN {X 0,Y 289.167,Z 548.553,A -85,B 0,C 180,E1 -17399.078,E2 -17399.078} C_VEL
LIN {X 0,Y 292.666,Z 536.116,A -85,B 0,C 180,E1 -17401.28,E2 -17401.28} C_VEL
LIN {X 0,Y 296.286,Z 522.505,A -85,B 0,C 180,E1 -17403.261,E2 -17403.261} C_VEL
LIN {X 0,Y 299.774,Z 508.082,A -85,B 0,C 180,E1 -17404.986,E2 -17404.986} C_VEL
LIN {X 0,Y 302.722,Z 494.753,A -85,B 0,C 180,E1 -17406.294,E2 -17406.294} C_VEL
LIN {X 0,Y 305.651,Z 479.314,A -85,B 0,C 180,E1 -17407.535,E2 -17407.535} C_VEL
LIN {X 0,Y 308.135,Z 463.525,A -85,B 0,C 180,E1 -17408.526,E2 -17408.526} C_VEL
LIN {X 0,Y 310.203,Z 447.451,A -85,B 0,C 180,E1 -17409.263,E2 -17409.263} C_VEL
LIN {X 0,Y 311.651,Z 431.041,A -85,B 0,C 180,E1 -17409.794,E2 -17409.794} C_VEL
LIN {X 0,Y 318.181,Z 296.796,A -85,B 0,C 180,E1 -17412.913,E2 -17412.913} C_VEL
LIN {X 0,Y 308.577,Z 276.909,A -85,B 0,C 180,E1 -17415.029,E2 -17415.029} C_VEL
LIN {X 0,Y 299.262,Z 259.778,A -85,B 0,C 180,E1 -17417.19,E2 -17417.19} C_VEL
LIN {X 0,Y 288.779,Z 242.153,A -85,B 0,C 180,E1 -17419.804,E2 -17419.804} C_VEL
LIN {X 0,Y 280.655,Z 229.909,A -85,B 0,C 180,E1 -17421.976,E2 -17421.976} C_VEL
LIN {X 0,Y 278.251,Z 226.025,A -85,B 0,C 180,E1 -17422.687,E2 -17422.687} C_VEL
LIN {X 0,Y 277.274,Z 223.239,A -85,B 0,C 180,E1 -17423.656,E2 -17423.656} C_VEL
LIN {X 0,Y 277.219,Z 223.242,A -85,B 0,C 180,E1 -17427.834,E2 -17427.834} C_VEL
LIN {X 0,Y 277.259,Z 223.263,A -85,B 0,C 180,E1 -17431.21,E2 -17431.21} C_VEL
LIN {X 0,Y 277.292,Z 223.231,A -85,B 0,C 180,E1 -17434.478,E2 -17434.478} C_VEL
LIN {X 0,Y 277.277,Z 223.256,A -85,B 0,C 180,E1 -17437.655,E2 -17437.655} C_VEL
LIN {X 0,Y 277.344,Z 223.215,A -85,B 0,C 180,E1 -17440.767,E2 -17440.767} C_VEL
LIN {X 0,Y 277.401,Z 223.229,A -85,B 0,C 180,E1 -17445.325,E2 -17445.325} C_VEL
LIN {X 0,Y 277.479,Z 223.208,A -85,B 0,C 180,E1 -17449.788,E2 -17449.788} C_VEL
LIN {X 0,Y 277.622,Z 223.212,A -85,B 0,C 180,E1 -17452.729,E2 -17452.729} C_VEL
LIN {X 0,Y 277.794,Z 223.168,A -85,B 0,C 180,E1 -17458.551,E2 -17458.551} C_VEL
LIN {X 0,Y 277.793,Z 223.193,A -85,B 0,C 180,E1 -17461.45,E2 -17461.45} C_VEL
LIN {X 0,Y 277.613,Z 223.214,A -85,B 0,C 180,E1 -17467.273,E2 -17467.273} C_VEL
LIN {X 0,Y 277.434,Z 223.217,A -85,B 0,C 180,E1 -17470.215,E2 -17470.215} C_VEL
LIN {X 0,Y 277.402,Z 223.239,A -85,B 0,C 180,E1 -17474.677,E2 -17474.677} C_VEL
LIN {X 0,Y 277.32,Z 223.222,A -85,B 0,C 180,E1 -17479.236,E2 -17479.236} C_VEL
LIN {X 0,Y 277.295,Z 223.242,A -85,B 0,C 180,E1 -17484.172,E2 -17484.172} C_VEL
LIN {X 0,Y 277.302,Z 223.238,A -85,B 0,C 180,E1 -17487.507,E2 -17487.507} C_VEL
LIN {X 0,Y 277.252,Z 223.257,A -85,B 0,C 180,E1 -17490.485,E2 -17490.485} C_VEL
LIN {X 0,Y 277.227,Z 223.243,A -85,B 0,C 180,E1 -17493.899,E2 -17493.899} C_VEL
LIN {X 0,Y 277.246,Z 223.253,A -85,B 0,C 180,E1 -17497.474,E2 -17497.474} C_VEL
LIN {X 0,Y 277.193,Z 223.264,A -85,B 0,C 180,E1 -17501.241,E2 -17501.241} C_VEL
LIN {X 0,Y 277.186,Z 223.247,A -85,B 0,C 180,E1 -17505.231,E2 -17505.231} C_VEL
LIN {X 0,Y 277.209,Z 223.254,A -85,B 0,C 180,E1 -17509.517,E2 -17509.517} C_VEL
LIN {X 0,Y 277.25,Z 223.261,A -85,B 0,C 180,E1 -17512.534,E2 -17512.534} C_VEL
LIN {X 0,Y 277.237,Z 223.247,A -85,B 0,C 180,E1 -17516.109,E2 -17516.109} C_VEL
LIN {X 0,Y 277.254,Z 223.248,A -85,B 0,C 180,E1 -17519.543,E2 -17519.543} C_VEL
LIN {X 0,Y 277.286,Z 223.253,A -85,B 0,C 180,E1 -17522.861,E2 -17522.861} C_VEL
LIN {X 0,Y 277.231,Z 223.26,A -85,B 0,C 180,E1 -17524.509,E2 -17524.509} C_VEL
LIN {X 0,Y 278.086,Z 225.838,A -85,B 0,C 180,E1 -17524.807,E2 -17524.807} C_VEL
LIN {X 0,Y 280.163,Z 228.142,A -85,B 0,C 180,E1 -17525.362,E2 -17525.362} C_VEL
LIN {X 0,Y 281.034,Z 229.485,A -85,B 0,C 180,E1 -17525.608,E2 -17525.608} C_VEL
LIN {X 0,Y 283.402,Z 232.696,A -85,B 0,C 180,E1 -17526.247,E2 -17526.247} C_VEL
LIN {X 0,Y 286.678,Z 237.276,A -85,B 0,C 180,E1 -17527.107,E2 -17527.107} C_VEL
LIN {X 0,Y 295.906,Z 250.828,A -85,B 0,C 180,E1 -17529.397,E2 -17529.397} C_VEL
LIN {X 0,Y 305.178,Z 265.343,A -85,B 0,C 180,E1 -17531.539,E2 -17531.539} C_VEL
LIN {X 0,Y 315.129,Z 282.489,A -85,B 0,C 180,E1 -17533.691,E2 -17533.691} C_VEL
LIN {X 0,Y 318.301,Z 288.957,A -85,B 0,C 180,E1 -17534.371,E2 -17534.371} C_VEL
LIN {X 0,Y 311.788,Z 420.44,A -85,B 0,C 180,E1 -17537.432,E2 -17537.432} C_VEL
LIN {X 0,Y 310.172,Z 437.552,A -85,B 0,C 180,E1 -17538.071,E2 -17538.071} C_VEL
LIN {X 0,Y 308.16,Z 453.37,A -85,B 0,C 180,E1 -17538.909,E2 -17538.909} C_VEL
LIN {X 0,Y 305.868,Z 468.028,A -85,B 0,C 180,E1 -17539.913,E2 -17539.913} C_VEL
LIN {X 0,Y 303.147,Z 482.765,A -85,B 0,C 180,E1 -17541.169,E2 -17541.169} C_VEL
LIN {X 0,Y 299.867,Z 497.898,A -85,B 0,C 180,E1 -17542.767,E2 -17542.767} C_VEL
LIN {X 0,Y 296.407,Z 511.809,A -85,B 0,C 180,E1 -17544.561,E2 -17544.561} C_VEL
LIN {X 0,Y 293.028,Z 524.63,A -85,B 0,C 180,E1 -17546.566,E2 -17546.566} C_VEL
LIN {X 0,Y 289.967,Z 535.681,A -85,B 0,C 180,E1 -17548.615,E2 -17548.615} C_VEL
LIN {X 0,Y 286.73,Z 546.764,A -85,B 0,C 180,E1 -17551.057,E2 -17551.057} C_VEL
LIN {X 0,Y 283.582,Z 557.42,A -85,B 0,C 180,E1 -17553.911,E2 -17553.911} C_VEL
LIN {X 0,Y 280.931,Z 566.352,A -85,B 0,C 180,E1 -17556.828,E2 -17556.828} C_VEL
LIN {X 0,Y 279.175,Z 572.942,A -85,B 0,C 180,E1 -17559.421,E2 -17559.421} C_VEL
LIN {X 0,Y 277.569,Z 579.237,A -85,B 0,C 180,E1 -17562.431,E2 -17562.431} C_VEL
LIN {X 0,Y 276.579,Z 583.639,A -85,B 0,C 180,E1 -17565.069,E2 -17565.069} C_VEL
LIN {X 0,Y 275.801,Z 587.302,A -85,B 0,C 180,E1 -17567.808,E2 -17567.808} C_VEL
LIN {X 0,Y 275.185,Z 590.342,A -85,B 0,C 180,E1 -17570.953,E2 -17570.953} C_VEL
LIN {X 0,Y 274.871,Z 592.312,A -85,B 0,C 180,E1 -17574.151,E2 -17574.151} C_VEL
LIN {X 0,Y 274.852,Z 593.088,A -85,B 0,C 180,E1 -17577.407,E2 -17577.407} C_VEL
LIN {X 0,Y 274.96,Z 592.973,A -85,B 0,C 180,E1 -17579.651,E2 -17579.651} C_VEL
LIN {X 0,Y 275.185,Z 591.928,A -85,B 0,C 180,E1 -17582.562,E2 -17582.562} C_VEL
LIN {X 0,Y 275.763,Z 589.65,A -85,B 0,C 180,E1 -17585.888,E2 -17585.888} C_VEL
LIN {X 0,Y 276.401,Z 587.536,A -85,B 0,C 180,E1 -17587.978,E2 -17587.978} C_VEL
LIN {X 0,Y 277.633,Z 583.349,A -85,B 0,C 180,E1 -17591.163,E2 -17591.163} C_VEL
LIN {X 0,Y 279.06,Z 578.772,A -85,B 0,C 180,E1 -17593.836,E2 -17593.836} C_VEL
LIN {X 0,Y 281.357,Z 571.847,A -85,B 0,C 180,E1 -17597.1,E2 -17597.1} C_VEL
LIN {X 0,Y 284.208,Z 564.024,A -85,B 0,C 180,E1 -17600.05,E2 -17600.05} C_VEL
LIN {X 0,Y 287.432,Z 555.083,A -85,B 0,C 180,E1 -17602.8,E2 -17602.8} C_VEL
LIN {X 0,Y 290.828,Z 545.544,A -85,B 0,C 180,E1 -17605.251,E2 -17605.251} C_VEL
LIN {X 0,Y 294.566,Z 534.793,A -85,B 0,C 180,E1 -17607.568,E2 -17607.568} C_VEL
LIN {X 0,Y 298.724,Z 522.066,A -85,B 0,C 180,E1 -17609.84,E2 -17609.84} C_VEL
LIN {X 0,Y 302.929,Z 508.327,A -85,B 0,C 180,E1 -17611.839,E2 -17611.839} C_VEL
LIN {X 0,Y 306.51,Z 495.251,A -85,B 0,C 180,E1 -17613.413,E2 -17613.413} C_VEL
LIN {X 0,Y 307.947,Z 489.581,A -85,B 0,C 180,E1 -17614.016,E2 -17614.016} C_VEL
LIN {X 0,Y 308.783,Z 484.56,A -85,B 0,C 180,E1 -17614.575,E2 -17614.575} C_VEL
LIN {X 0,Y 308.478,Z 476.536,A -85,B 0,C 180,E1 -17615.657,E2 -17615.657} C_VEL
LIN {X 0,Y 308.092,Z 468.336,A -85,B 0,C 180,E1 -17616.686,E2 -17616.686} C_VEL
LIN {X 0,Y 308.567,Z 463.04,A -85,B 0,C 180,E1 -17617.16,E2 -17617.16} C_VEL
LIN {X 0,Y 311.291,Z 446.842,A -85,B 0,C 180,E1 -17618.148,E2 -17618.148} C_VEL
LIN {X 0,Y 313.445,Z 430.527,A -85,B 0,C 180,E1 -17618.877,E2 -17618.877} C_VEL
LIN {X 0,Y 314.994,Z 413.167,A -85,B 0,C 180,E1 -17619.392,E2 -17619.392} C_VEL
LIN {X 0,Y 321.962,Z 296.592,A -85,B 0,C 180,E1 -17622.146,E2 -17622.146} C_VEL
LIN {X 0,Y 317.075,Z 286.993,A -85,B 0,C 180,E1 -17623.597,E2 -17623.597} C_VEL
LIN {X 0,Y 310.196,Z 275.529,A -85,B 0,C 180,E1 -17625.751,E2 -17625.751} C_VEL
LIN {X 0,Y 304.642,Z 267.204,A -85,B 0,C 180,E1 -17627.648,E2 -17627.648} C_VEL
LIN {X 0,Y 299.63,Z 260.038,A -85,B 0,C 180,E1 -17629.542,E2 -17629.542} C_VEL
LIN {X 0,Y 296.438,Z 255.749,A -85,B 0,C 180,E1 -17630.838,E2 -17630.838} C_VEL
LIN {X 0,Y 292.891,Z 251.035,A -85,B 0,C 180,E1 -17632.416,E2 -17632.416} C_VEL
LIN {X 0,Y 290.179,Z 247.352,A -85,B 0,C 180,E1 -17633.742,E2 -17633.742} C_VEL
LIN {X 0,Y 289.514,Z 246.515,A -85,B 0,C 180,E1 -17634.078,E2 -17634.078} C_VEL
LIN {X 0,Y 286.743,Z 243.623,A -85,B 0,C 180,E1 -17635.504,E2 -17635.504} C_VEL
LIN {X 0,Y 285.446,Z 241.529,A -85,B 0,C 180,E1 -17636.294,E2 -17636.294} C_VEL
LIN {X 0,Y 282.993,Z 239.302,A -85,B 0,C 180,E1 -17637.775,E2 -17637.775} C_VEL
LIN {X 0,Y 281.159,Z 235.908,A -85,B 0,C 180,E1 -17639.124,E2 -17639.124} C_VEL
LIN {X 0,Y 278.091,Z 233.717,A -85,B 0,C 180,E1 -17641.447,E2 -17641.447} C_VEL
LIN {X 0,Y 276.536,Z 231.14,A -85,B 0,C 180,E1 -17643.004,E2 -17643.004} C_VEL
LIN {X 0,Y 276.147,Z 230.173,A -85,B 0,C 180,E1 -17643.465,E2 -17643.465} C_VEL
LIN {X 0,Y 273.128,Z 228.717,A -85,B 0,C 180,E1 -17647.205,E2 -17647.205} C_VEL
LIN {X 0,Y 271.601,Z 227.26,A -85,B 0,C 180,E1 -17651.114,E2 -17651.114} C_VEL
LIN {X 0,Y 271.401,Z 227.03,A -85,B 0,C 180,E1 -17654.24,E2 -17654.24} C_VEL
LIN {X 0,Y 272.525,Z 228.503,A -85,B 0,C 180,E1 -17658.415,E2 -17658.415} C_VEL
LIN {X 0,Y 275.893,Z 230.369,A -85,B 0,C 180,E1 -17662.958,E2 -17662.958} C_VEL
LIN {X 0,Y 277.019,Z 233.02,A -85,B 0,C 180,E1 -17664.255,E2 -17664.255} C_VEL
LIN {X 0,Y 279.172,Z 235.185,A -85,B 0,C 180,E1 -17666.138,E2 -17666.138} C_VEL
LIN {X 0,Y 280.86,Z 236.211,A -85,B 0,C 180,E1 -17667.349,E2 -17667.349} C_VEL
LIN {X 0,Y 282.56,Z 239.238,A -85,B 0,C 180,E1 -17668.606,E2 -17668.606} C_VEL
LIN {X 0,Y 285.585,Z 242.149,A -85,B 0,C 180,E1 -17670.455,E2 -17670.455} C_VEL
LIN {X 0,Y 287.943,Z 245.503,A -85,B 0,C 180,E1 -17671.8,E2 -17671.8} C_VEL
LIN {X 0,Y 291.714,Z 250.426,A -85,B 0,C 180,E1 -17673.711,E2 -17673.711} C_VEL
LIN {X 0,Y 295.873,Z 256.467,A -85,B 0,C 180,E1 -17675.633,E2 -17675.633} C_VEL
LIN {X 0,Y 300.725,Z 263.834,A -85,B 0,C 180,E1 -17677.631,E2 -17677.631} C_VEL
LIN {X 0,Y 305.876,Z 272.299,A -85,B 0,C 180,E1 -17679.572,E2 -17679.572} C_VEL
LIN {X 0,Y 311.516,Z 282.247,A -85,B 0,C 180,E1 -17681.507,E2 -17681.507} C_VEL
LIN {X 0,Y 317.554,Z 293.936,A -85,B 0,C 180,E1 -17683.415,E2 -17683.415} C_VEL
LIN {X 0,Y 321.703,Z 303.184,A -85,B 0,C 180,E1 -17684.673,E2 -17684.673} C_VEL
LIN {X 0,Y 317.624,Z 370.992,A -85,B 0,C 180,E1 -17686.266,E2 -17686.266} C_VEL
LIN {X 0,Y 313.761,Z 433.862,A -85,B 0,C 180,E1 -17687.778,E2 -17687.778} C_VEL
LIN {X 0,Y 311.673,Z 451.35,A -85,B 0,C 180,E1 -17688.403,E2 -17688.403} C_VEL
LIN {X 0,Y 308.899,Z 468.12,A -85,B 0,C 180,E1 -17689.253,E2 -17689.253} C_VEL
LIN {X 0,Y 305.582,Z 484.267,A -85,B 0,C 180,E1 -17690.339,E2 -17690.339} C_VEL
LIN {X 0,Y 301.871,Z 499.854,A -85,B 0,C 180,E1 -17691.691,E2 -17691.691} C_VEL
LIN {X 0,Y 298.099,Z 513.453,A -85,B 0,C 180,E1 -17693.127,E2 -17693.127} C_VEL
LIN {X 0,Y 293.804,Z 527.579,A -85,B 0,C 180,E1 -17694.961,E2 -17694.961} C_VEL
LIN {X 0,Y 289.697,Z 539.909,A -85,B 0,C 180,E1 -17696.915,E2 -17696.915} C_VEL
LIN {X 0,Y 285.444,Z 552.092,A -85,B 0,C 180,E1 -17699.236,E2 -17699.236} C_VEL
LIN {X 0,Y 281.63,Z 562.823,A -85,B 0,C 180,E1 -17701.694,E2 -17701.694} C_VEL
LIN {X 0,Y 277.864,Z 573.116,A -85,B 0,C 180,E1 -17704.531,E2 -17704.531} C_VEL
LIN {X 0,Y 274.786,Z 581.722,A -85,B 0,C 180,E1 -17707.438,E2 -17707.438} C_VEL
LIN {X 0,Y 272.392,Z 588.928,A -85,B 0,C 180,E1 -17710.399,E2 -17710.399} C_VEL
LIN {X 0,Y 270.583,Z 594.952,A -85,B 0,C 180,E1 -17713.396,E2 -17713.396} C_VEL
LIN {X 0,Y 269.116,Z 600.823,A -85,B 0,C 180,E1 -17717.172,E2 -17717.172} C_VEL
LIN {X 0,Y 268.309,Z 605.017,A -85,B 0,C 180,E1 -17720.954,E2 -17720.954} C_VEL
LIN {X 0,Y 268.129,Z 607.703,A -85,B 0,C 180,E1 -17724.885,E2 -17724.885} C_VEL
LIN {X 0,Y 268.146,Z 608.472,A -85,B 0,C 180,E1 -17726.992,E2 -17726.992} C_VEL
LIN {X 0,Y 268.199,Z 608.683,A -85,B 0,C 180,E1 -17729.996,E2 -17729.996} C_VEL
LIN {X 0,Y 268.156,Z 607.984,A -85,B 0,C 180,E1 -17733.001,E2 -17733.001} C_VEL
LIN {X 0,Y 268.134,Z 606.195,A -85,B 0,C 180,E1 -17736.014,E2 -17736.014} C_VEL
LIN {X 0,Y 268.303,Z 603.467,A -85,B 0,C 180,E1 -17739.038,E2 -17739.038} C_VEL
LIN {X 0,Y 269.035,Z 598.482,A -85,B 0,C 180,E1 -17742.825,E2 -17742.825} C_VEL
LIN {X 0,Y 270.047,Z 593.537,A -85,B 0,C 180,E1 -17745.653,E2 -17745.653} C_VEL
LIN {X 0,Y 271.649,Z 586.637,A -85,B 0,C 180,E1 -17748.864,E2 -17748.864} C_VEL
LIN {X 0,Y 273.813,Z 578.763,A -85,B 0,C 180,E1 -17751.845,E2 -17751.845} C_VEL
LIN {X 0,Y 276.556,Z 569.242,A -85,B 0,C 180,E1 -17754.786,E2 -17754.786} C_VEL
LIN {X 0,Y 279.545,Z 559.412,A -85,B 0,C 180,E1 -17757.306,E2 -17757.306} C_VEL
LIN {X 0,Y 282.871,Z 547.912,A -85,B 0,C 180,E1 -17759.79,E2 -17759.79} C_VEL
LIN {X 0,Y 286.526,Z 535.39,A -85,B 0,C 180,E1 -17762.029,E2 -17762.029} C_VEL
LIN {X 0,Y 290.314,Z 521.729,A -85,B 0,C 180,E1 -17764.038,E2 -17764.038} C_VEL
LIN {X 0,Y 293.628,Z 508.311,A -85,B 0,C 180,E1 -17765.664,E2 -17765.664} C_VEL
LIN {X 0,Y 296.575,Z 495.465,A -85,B 0,C 180,E1 -17766.959,E2 -17766.959} C_VEL
LIN {X 0,Y 299.586,Z 480.257,A -85,B 0,C 180,E1 -17768.218,E2 -17768.218} C_VEL
LIN {X 0,Y 302.345,Z 463.363,A -85,B 0,C 180,E1 -17769.297,E2 -17769.297} C_VEL
LIN {X 0,Y 304.466,Z 447.309,A -85,B 0,C 180,E1 -17770.043,E2 -17770.043} C_VEL
LIN {X 0,Y 305.96,Z 431.04,A -85,B 0,C 180,E1 -17770.576,E2 -17770.576} C_VEL
LIN {X 0,Y 312.666,Z 299.259,A -85,B 0,C 180,E1 -17773.672,E2 -17773.672} C_VEL
LIN {X 0,Y 303.135,Z 279.521,A -85,B 0,C 180,E1 -17775.844,E2 -17775.844} C_VEL
LIN {X 0,Y 294.019,Z 262.768,A -85,B 0,C 180,E1 -17778.044,E2 -17778.044} C_VEL
LIN {X 0,Y 284.642,Z 246.929,A -85,B 0,C 180,E1 -17780.465,E2 -17780.465} C_VEL
LIN {X 0,Y 277.059,Z 235.357,A -85,B 0,C 180,E1 -17782.556,E2 -17782.556} C_VEL
LIN {X 0,Y 273.966,Z 230.646,A -85,B 0,C 180,E1 -17783.462,E2 -17783.462} C_VEL
LIN {X 0,Y 270.575,Z 225.645,A -85,B 0,C 180,E1 -17784.529,E2 -17784.529} C_VEL
LIN {X 0,Y 270.172,Z 224.138,A -85,B 0,C 180,E1 -17785.091,E2 -17785.091} C_VEL
LIN {X 0,Y 270.176,Z 224.124,A -85,B 0,C 180,E1 -17789.129,E2 -17789.129} C_VEL
LIN {X 0,Y 270.239,Z 224.119,A -85,B 0,C 180,E1 -17792.144,E2 -17792.144} C_VEL
LIN {X 0,Y 270.257,Z 224.12,A -85,B 0,C 180,E1 -17795.516,E2 -17795.516} C_VEL
LIN {X 0,Y 270.3,Z 224.091,A -85,B 0,C 180,E1 -17800.245,E2 -17800.245} C_VEL
LIN {X 0,Y 270.369,Z 224.111,A -85,B 0,C 180,E1 -17804.934,E2 -17804.934} C_VEL
LIN {X 0,Y 270.414,Z 224.082,A -85,B 0,C 180,E1 -17809.519,E2 -17809.519} C_VEL
LIN {X 0,Y 270.581,Z 224.091,A -85,B 0,C 180,E1 -17812.539,E2 -17812.539} C_VEL
LIN {X 0,Y 270.759,Z 224.041,A -85,B 0,C 180,E1 -17818.513,E2 -17818.513} C_VEL
LIN {X 0,Y 270.759,Z 224.069,A -85,B 0,C 180,E1 -17821.488,E2 -17821.488} C_VEL
LIN {X 0,Y 270.571,Z 224.092,A -85,B 0,C 180,E1 -17827.463,E2 -17827.463} C_VEL
LIN {X 0,Y 270.386,Z 224.091,A -85,B 0,C 180,E1 -17830.484,E2 -17830.484} C_VEL
LIN {X 0,Y 270.371,Z 224.117,A -85,B 0,C 180,E1 -17835.067,E2 -17835.067} C_VEL
LIN {X 0,Y 270.277,Z 224.102,A -85,B 0,C 180,E1 -17839.758,E2 -17839.758} C_VEL
LIN {X 0,Y 270.251,Z 224.113,A -85,B 0,C 180,E1 -17844.589,E2 -17844.589} C_VEL
LIN {X 0,Y 270.251,Z 224.123,A -85,B 0,C 180,E1 -17847.912,E2 -17847.912} C_VEL
LIN {X 0,Y 270.164,Z 224.128,A -85,B 0,C 180,E1 -17851.352,E2 -17851.352} C_VEL
LIN {X 0,Y 270.182,Z 224.134,A -85,B 0,C 180,E1 -17854.909,E2 -17854.909} C_VEL
LIN {X 0,Y 270.181,Z 224.118,A -85,B 0,C 180,E1 -17858.714,E2 -17858.714} C_VEL
LIN {X 0,Y 270.15,Z 224.142,A -85,B 0,C 180,E1 -17863.253,E2 -17863.253} C_VEL
LIN {X 0,Y 270.158,Z 224.145,A -85,B 0,C 180,E1 -17867.446,E2 -17867.446} C_VEL
LIN {X 0,Y 270.196,Z 224.125,A -85,B 0,C 180,E1 -17871.379,E2 -17871.379} C_VEL
LIN {X 0,Y 270.191,Z 224.123,A -85,B 0,C 180,E1 -17875.099,E2 -17875.099} C_VEL
LIN {X 0,Y 270.176,Z 224.133,A -85,B 0,C 180,E1 -17879.141,E2 -17879.141} C_VEL
LIN {X 0,Y 270.241,Z 224.13,A -85,B 0,C 180,E1 -17882.889,E2 -17882.889} C_VEL
LIN {X 0,Y 271.117,Z 226.794,A -85,B 0,C 180,E1 -17883.22,E2 -17883.22} C_VEL
LIN {X 0,Y 273.256,Z 229.132,A -85,B 0,C 180,E1 -17883.83,E2 -17883.83} C_VEL
LIN {X 0,Y 275.924,Z 233.098,A -85,B 0,C 180,E1 -17884.611,E2 -17884.611} C_VEL
LIN {X 0,Y 277.375,Z 234.875,A -85,B 0,C 180,E1 -17885.011,E2 -17885.011} C_VEL
LIN {X 0,Y 287.157,Z 248.832,A -85,B 0,C 180,E1 -17887.636,E2 -17887.636} C_VEL
LIN {X 0,Y 296.514,Z 262.989,A -85,B 0,C 180,E1 -17889.935,E2 -17889.935} C_VEL
LIN {X 0,Y 305.98,Z 278.739,A -85,B 0,C 180,E1 -17892.113,E2 -17892.113} C_VEL
LIN {X 0,Y 311.726,Z 289.386,A -85,B 0,C 180,E1 -17893.377,E2 -17893.377} C_VEL
LIN {X 0,Y 312.794,Z 291.612,A -85,B 0,C 180,E1 -17893.613,E2 -17893.613} C_VEL
LIN {X 0,Y 306.103,Z 420.576,A -85,B 0,C 180,E1 -17896.646,E2 -17896.646} C_VEL
LIN {X 0,Y 304.449,Z 437.676,A -85,B 0,C 180,E1 -17897.293,E2 -17897.293} C_VEL
LIN {X 0,Y 302.355,Z 453.656,A -85,B 0,C 180,E1 -17898.151,E2 -17898.151} C_VEL
LIN {X 0,Y 299.917,Z 468.681,A -85,B 0,C 180,E1 -17899.199,E2 -17899.199} C_VEL
LIN {X 0,Y 297.104,Z 483.332,A -85,B 0,C 180,E1 -17900.472,E2 -17900.472} C_VEL
LIN {X 0,Y 293.707,Z 498.441,A -85,B 0,C 180,E1 -17902.095,E2 -17902.095} C_VEL
LIN {X 0,Y 290.086,Z 512.485,A -85,B 0,C 180,E1 -17903.947,E2 -17903.947} C_VEL
LIN {X 0,Y 286.924,Z 524.081,A -85,B 0,C 180,E1 -17905.789,E2 -17905.789} C_VEL
LIN {X 0,Y 283.695,Z 535.27,A -85,B 0,C 180,E1 -17907.874,E2 -17907.874} C_VEL
LIN {X 0,Y 280.334,Z 546.397,A -85,B 0,C 180,E1 -17910.363,E2 -17910.363} C_VEL
LIN {X 0,Y 277.384,Z 555.899,A -85,B 0,C 180,E1 -17912.908,E2 -17912.908} C_VEL
LIN {X 0,Y 274.553,Z 565.138,A -85,B 0,C 180,E1 -17915.88,E2 -17915.88} C_VEL
LIN {X 0,Y 272.352,Z 572.853,A -85,B 0,C 180,E1 -17918.91,E2 -17918.91} C_VEL
LIN {X 0,Y 270.681,Z 579.177,A -85,B 0,C 180,E1 -17921.992,E2 -17921.992} C_VEL
LIN {X 0,Y 269.441,Z 584.342,A -85,B 0,C 180,E1 -17925.18,E2 -17925.18} C_VEL
LIN {X 0,Y 268.59,Z 588.239,A -85,B 0,C 180,E1 -17928.303,E2 -17928.303} C_VEL
LIN {X 0,Y 267.996,Z 591.06,A -85,B 0,C 180,E1 -17931.542,E2 -17931.542} C_VEL
LIN {X 0,Y 267.746,Z 592.745,A -85,B 0,C 180,E1 -17934.836,E2 -17934.836} C_VEL
LIN {X 0,Y 267.772,Z 593.325,A -85,B 0,C 180,E1 -17938.195,E2 -17938.195} C_VEL
LIN {X 0,Y 267.876,Z 593.141,A -85,B 0,C 180,E1 -17940.025,E2 -17940.025} C_VEL
LIN {X 0,Y 268.179,Z 591.832,A -85,B 0,C 180,E1 -17943.393,E2 -17943.393} C_VEL
LIN {X 0,Y 268.972,Z 589.166,A -85,B 0,C 180,E1 -17946.942,E2 -17946.942} C_VEL
LIN {X 0,Y 269.876,Z 586.243,A -85,B 0,C 180,E1 -17949.647,E2 -17949.647} C_VEL
LIN {X 0,Y 271.823,Z 580.341,A -85,B 0,C 180,E1 -17953.618,E2 -17953.618} C_VEL
LIN {X 0,Y 274.493,Z 572.762,A -85,B 0,C 180,E1 -17957.403,E2 -17957.403} C_VEL
LIN {X 0,Y 277.21,Z 565.596,A -85,B 0,C 180,E1 -17960.219,E2 -17960.219} C_VEL
LIN {X 0,Y 280.54,Z 556.919,A -85,B 0,C 180,E1 -17963.04,E2 -17963.04} C_VEL
LIN {X 0,Y 283.936,Z 547.878,A -85,B 0,C 180,E1 -17965.507,E2 -17965.507} C_VEL
LIN {X 0,Y 288.215,Z 536.185,A -85,B 0,C 180,E1 -17968.131,E2 -17968.131} C_VEL
LIN {X 0,Y 292.257,Z 524.41,A -85,B 0,C 180,E1 -17970.312,E2 -17970.312} C_VEL
LIN {X 0,Y 296.553,Z 511.111,A -85,B 0,C 180,E1 -17972.347,E2 -17972.347} C_VEL
LIN {X 0,Y 300.499,Z 497.533,A -85,B 0,C 180,E1 -17974.064,E2 -17974.064} C_VEL
LIN {X 0,Y 304.166,Z 483.417,A -85,B 0,C 180,E1 -17975.531,E2 -17975.531} C_VEL
LIN {X 0,Y 307.745,Z 467.343,A -85,B 0,C 180,E1 -17976.861,E2 -17976.861} C_VEL
LIN {X 0,Y 308.567,Z 463.04,A -85,B 0,C 180,E1 -17977.16,E2 -17977.16} C_VEL
LIN {X 0,Y 309.13,Z 457.661,A -85,B 0,C 180,E1 -17977.607,E2 -17977.607} C_VEL
LIN {X 0,Y 307.929,Z 442.013,A -85,B 0,C 180,E1 -17979.185,E2 -17979.185} C_VEL
LIN {X 0,Y 307.915,Z 436.512,A -85,B 0,C 180,E1 -17979.58,E2 -17979.58} C_VEL
LIN {X 0,Y 308.076,Z 434.622,A -85,B 0,C 180,E1 -17979.674,E2 -17979.674} C_VEL
LIN {X 0,Y 309.858,Z 417.358,A -85,B 0,C 180,E1 -17980.243,E2 -17980.243} C_VEL
LIN {X 0,Y 317.387,Z 299.684,A -85,B 0,C 180,E1 -17983.037,E2 -17983.037} C_VEL
LIN {X 0,Y 313.081,Z 291.221,A -85,B 0,C 180,E1 -17984.372,E2 -17984.372} C_VEL
LIN {X 0,Y 305.88,Z 279.183,A -85,B 0,C 180,E1 -17986.752,E2 -17986.752} C_VEL
LIN {X 0,Y 300.056,Z 270.257,A -85,B 0,C 180,E1 -17988.893,E2 -17988.893} C_VEL
LIN {X 0,Y 294.368,Z 262.207,A -85,B 0,C 180,E1 -17991.227,E2 -17991.227} C_VEL
LIN {X 0,Y 291.292,Z 257.986,A -85,B 0,C 180,E1 -17992.635,E2 -17992.635} C_VEL
LIN {X 0,Y 288.098,Z 253.737,A -85,B 0,C 180,E1 -17994.226,E2 -17994.226} C_VEL
LIN {X 0,Y 284.493,Z 249.491,A -85,B 0,C 180,E1 -17996.193,E2 -17996.193} C_VEL
LIN {X 0,Y 283.822,Z 248.256,A -85,B 0,C 180,E1 -17996.628,E2 -17996.628} C_VEL
LIN {X 0,Y 281.26,Z 245.807,A -85,B 0,C 180,E1 -17998.227,E2 -17998.227} C_VEL
LIN {X 0,Y 279.524,Z 242.665,A -85,B 0,C 180,E1 -17999.545,E2 -17999.545} C_VEL
LIN {X 0,Y 276.672,Z 240.431,A -85,B 0,C 180,E1 -18001.819,E2 -18001.819} C_VEL
LIN {X 0,Y 275.065,Z 237.653,A -85,B 0,C 180,E1 -18003.501,E2 -18003.501} C_VEL
LIN {X 0,Y 274.729,Z 237.101,A -85,B 0,C 180,E1 -18003.884,E2 -18003.884} C_VEL
LIN {X 0,Y 271.34,Z 235.03,A -85,B 0,C 180,E1 -18008.76,E2 -18008.76} C_VEL
LIN {X 0,Y 270.497,Z 234.067,A -85,B 0,C 180,E1 -18011.996,E2 -18011.996} C_VEL
LIN {X 0,Y 270.449,Z 234.065,A -85,B 0,C 180,E1 -18014.292,E2 -18014.292} C_VEL
LIN {X 0,Y 272.427,Z 236.227,A -85,B 0,C 180,E1 -18019.901,E2 -18019.901} C_VEL
LIN {X 0,Y 274.576,Z 237.345,A -85,B 0,C 180,E1 -18022.631,E2 -18022.631} C_VEL
LIN {X 0,Y 275.813,Z 239.973,A -85,B 0,C 180,E1 -18024.059,E2 -18024.059} C_VEL
LIN {X 0,Y 278.059,Z 242.195,A -85,B 0,C 180,E1 -18026.049,E2 -18026.049} C_VEL
LIN {X 0,Y 279.299,Z 243.074,A -85,B 0,C 180,E1 -18026.98,E2 -18026.98} C_VEL
LIN {X 0,Y 281.265,Z 246.288,A -85,B 0,C 180,E1 -18028.444,E2 -18028.444} C_VEL
LIN {X 0,Y 283.782,Z 248.679,A -85,B 0,C 180,E1 -18030.015,E2 -18030.015} C_VEL
LIN {X 0,Y 286.316,Z 252.275,A -85,B 0,C 180,E1 -18031.514,E2 -18031.514} C_VEL
LIN {X 0,Y 289.456,Z 256.585,A -85,B 0,C 180,E1 -18033.162,E2 -18033.162} C_VEL
LIN {X 0,Y 293.582,Z 262.745,A -85,B 0,C 180,E1 -18035.15,E2 -18035.15} C_VEL
LIN {X 0,Y 298.018,Z 269.662,A -85,B 0,C 180,E1 -18037.051,E2 -18037.051} C_VEL
LIN {X 0,Y 302.857,Z 277.839,A -85,B 0,C 180,E1 -18038.956,E2 -18038.956} C_VEL
LIN {X 0,Y 308.98,Z 288.877,A -85,B 0,C 180,E1 -18041.132,E2 -18041.132} C_VEL
LIN {X 0,Y 314.383,Z 299.985,A -85,B 0,C 180,E1 -18042.917,E2 -18042.917} C_VEL
LIN {X 0,Y 317.059,Z 305.994,A -85,B 0,C 180,E1 -18043.764,E2 -18043.764} C_VEL
LIN {X 0,Y 309.002,Z 433.031,A -85,B 0,C 180,E1 -18046.807,E2 -18046.807} C_VEL
LIN {X 0,Y 306.891,Z 450.365,A -85,B 0,C 180,E1 -18047.418,E2 -18047.418} C_VEL
LIN {X 0,Y 304.324,Z 465.679,A -85,B 0,C 180,E1 -18048.175,E2 -18048.175} C_VEL
LIN {X 0,Y 301.119,Z 481.318,A -85,B 0,C 180,E1 -18049.191,E2 -18049.191} C_VEL
LIN {X 0,Y 297.658,Z 495.832,A -85,B 0,C 180,E1 -18050.392,E2 -18050.392} C_VEL
LIN {X 0,Y 293.36,Z 511.006,A -85,B 0,C 180,E1 -18051.952,E2 -18051.952} C_VEL
LIN {X 0,Y 289.032,Z 524.982,A -85,B 0,C 180,E1 -18053.739,E2 -18053.739} C_VEL
LIN {X 0,Y 284.471,Z 538.274,A -85,B 0,C 180,E1 -18055.8,E2 -18055.8} C_VEL
LIN {X 0,Y 280.53,Z 549.21,A -85,B 0,C 180,E1 -18057.832,E2 -18057.832} C_VEL
LIN {X 0,Y 276.471,Z 560.125,A -85,B 0,C 180,E1 -18060.281,E2 -18060.281} C_VEL
LIN {X 0,Y 272.794,Z 569.503,A -85,B 0,C 180,E1 -18062.785,E2 -18062.785} C_VEL
LIN {X 0,Y 269.674,Z 577.667,A -85,B 0,C 180,E1 -18065.353,E2 -18065.353} C_VEL
LIN {X 0,Y 266.85,Z 585.488,A -85,B 0,C 180,E1 -18068.36,E2 -18068.36} C_VEL
LIN {X 0,Y 264.593,Z 592.034,A -85,B 0,C 180,E1 -18071.41,E2 -18071.41} C_VEL
LIN {X 0,Y 262.988,Z 597.412,A -85,B 0,C 180,E1 -18074.497,E2 -18074.497} C_VEL
LIN {X 0,Y 261.882,Z 601.631,A -85,B 0,C 180,E1 -18077.599,E2 -18077.599} C_VEL
LIN {X 0,Y 261.239,Z 604.883,A -85,B 0,C 180,E1 -18080.708,E2 -18080.708} C_VEL
LIN {X 0,Y 261.034,Z 607.031,A -85,B 0,C 180,E1 -18083.814,E2 -18083.814} C_VEL
LIN {X 0,Y 261.039,Z 608.287,A -85,B 0,C 180,E1 -18086.91,E2 -18086.91} C_VEL
LIN {X 0,Y 261.125,Z 608.469,A -85,B 0,C 180,E1 -18089.996,E2 -18089.996} C_VEL
LIN {X 0,Y 261.069,Z 607.749,A -85,B 0,C 180,E1 -18093.082,E2 -18093.082} C_VEL
LIN {X 0,Y 261.031,Z 605.928,A -85,B 0,C 180,E1 -18096.179,E2 -18096.179} C_VEL
LIN {X 0,Y 261.23,Z 603.167,A -85,B 0,C 180,E1 -18099.285,E2 -18099.285} C_VEL
LIN {X 0,Y 262.035,Z 598.146,A -85,B 0,C 180,E1 -18103.174,E2 -18103.174} C_VEL
LIN {X 0,Y 263.19,Z 592.72,A -85,B 0,C 180,E1 -18106.313,E2 -18106.313} C_VEL
LIN {X 0,Y 264.838,Z 586.217,A -85,B 0,C 180,E1 -18109.368,E2 -18109.368} C_VEL
LIN {X 0,Y 267.124,Z 578.301,A -85,B 0,C 180,E1 -18112.421,E2 -18112.421} C_VEL
LIN {X 0,Y 270.002,Z 568.738,A -85,B 0,C 180,E1 -18115.43,E2 -18115.43} C_VEL
LIN {X 0,Y 273.144,Z 558.846,A -85,B 0,C 180,E1 -18118.001,E2 -18118.001} C_VEL
LIN {X 0,Y 276.61,Z 547.271,A -85,B 0,C 180,E1 -18120.535,E2 -18120.535} C_VEL
LIN {X 0,Y 280.421,Z 534.66,A -85,B 0,C 180,E1 -18122.812,E2 -18122.812} C_VEL
LIN {X 0,Y 284.36,Z 521.06,A -85,B 0,C 180,E1 -18124.83,E2 -18124.83} C_VEL
LIN {X 0,Y 287.481,Z 508.703,A -85,B 0,C 180,E1 -18126.353,E2 -18126.353} C_VEL
LIN {X 0,Y 290.47,Z 496.178,A -85,B 0,C 180,E1 -18127.651,E2 -18127.651} C_VEL
LIN {X 0,Y 293.762,Z 480.083,A -85,B 0,C 180,E1 -18129.007,E2 -18129.007} C_VEL
LIN {X 0,Y 296.606,Z 463.186,A -85,B 0,C 180,E1 -18130.099,E2 -18130.099} C_VEL
LIN {X 0,Y 298.79,Z 447.138,A -85,B 0,C 180,E1 -18130.852,E2 -18130.852} C_VEL
LIN {X 0,Y 300.375,Z 430.101,A -85,B 0,C 180,E1 -18131.413,E2 -18131.413} C_VEL
LIN {X 0,Y 307.091,Z 301.57,A -85,B 0,C 180,E1 -18134.475,E2 -18134.475} C_VEL
LIN {X 0,Y 298.435,Z 283.538,A -85,B 0,C 180,E1 -18136.522,E2 -18136.522} C_VEL
LIN {X 0,Y 290.288,Z 268.385,A -85,B 0,C 180,E1 -18138.548,E2 -18138.548} C_VEL
LIN {X 0,Y 280.895,Z 252.199,A -85,B 0,C 180,E1 -18141.052,E2 -18141.052} C_VEL
LIN {X 0,Y 273.137,Z 240.255,A -85,B 0,C 180,E1 -18143.257,E2 -18143.257} C_VEL
LIN {X 0,Y 269.125,Z 234.143,A -85,B 0,C 180,E1 -18144.477,E2 -18144.477} C_VEL
LIN {X 0,Y 265.942,Z 229.81,A -85,B 0,C 180,E1 -18145.463,E2 -18145.463} C_VEL
LIN {X 0,Y 263.98,Z 227.585,A -85,B 0,C 180,E1 -18146.074,E2 -18146.074} C_VEL
LIN {X 0,Y 263.184,Z 225.223,A -85,B 0,C 180,E1 -18146.467,E2 -18146.467} C_VEL
LIN {X 0,Y 263.142,Z 225.002,A -85,B 0,C 180,E1 -18146.804,E2 -18146.804} C_VEL
LIN {X 0,Y 263.154,Z 225.019,A -85,B 0,C 180,E1 -18151.268,E2 -18151.268} C_VEL
LIN {X 0,Y 263.204,Z 224.992,A -85,B 0,C 180,E1 -18155.198,E2 -18155.198} C_VEL
LIN {X 0,Y 263.263,Z 224.968,A -85,B 0,C 180,E1 -18159.694,E2 -18159.694} C_VEL
LIN {X 0,Y 263.318,Z 224.994,A -85,B 0,C 180,E1 -18164.521,E2 -18164.521} C_VEL
LIN {X 0,Y 263.347,Z 224.956,A -85,B 0,C 180,E1 -18169.234,E2 -18169.234} C_VEL
LIN {X 0,Y 263.542,Z 224.97,A -85,B 0,C 180,E1 -18172.338,E2 -18172.338} C_VEL
LIN {X 0,Y 263.724,Z 224.915,A -85,B 0,C 180,E1 -18178.474,E2 -18178.474} C_VEL
LIN {X 0,Y 263.724,Z 224.946,A -85,B 0,C 180,E1 -18181.528,E2 -18181.528} C_VEL
LIN {X 0,Y 263.531,Z 224.969,A -85,B 0,C 180,E1 -18187.664,E2 -18187.664} C_VEL
LIN {X 0,Y 263.326,Z 224.966,A -85,B 0,C 180,E1 -18190.768,E2 -18190.768} C_VEL
LIN {X 0,Y 263.32,Z 224.994,A -85,B 0,C 180,E1 -18195.481,E2 -18195.481} C_VEL
LIN {X 0,Y 263.24,Z 224.984,A -85,B 0,C 180,E1 -18200.309,E2 -18200.309} C_VEL
LIN {X 0,Y 263.186,Z 224.985,A -85,B 0,C 180,E1 -18205.295,E2 -18205.295} C_VEL
LIN {X 0,Y 263.159,Z 225.014,A -85,B 0,C 180,E1 -18208.733,E2 -18208.733} C_VEL
LIN {X 0,Y 263.113,Z 224.996,A -85,B 0,C 180,E1 -18212.292,E2 -18212.292} C_VEL
LIN {X 0,Y 263.163,Z 225.015,A -85,B 0,C 180,E1 -18216.767,E2 -18216.767} C_VEL
LIN {X 0,Y 263.089,Z 225.001,A -85,B 0,C 180,E1 -18219.877,E2 -18219.877} C_VEL
LIN {X 0,Y 263.089,Z 225.009,A -85,B 0,C 180,E1 -18223.993,E2 -18223.993} C_VEL
LIN {X 0,Y 263.111,Z 225.022,A -85,B 0,C 180,E1 -18228.411,E2 -18228.411} C_VEL
LIN {X 0,Y 263.147,Z 225.011,A -85,B 0,C 180,E1 -18232.107,E2 -18232.107} C_VEL
LIN {X 0,Y 263.142,Z 225.001,A -85,B 0,C 180,E1 -18235.89,E2 -18235.89} C_VEL
LIN {X 0,Y 263.13,Z 225.006,A -85,B 0,C 180,E1 -18240.394,E2 -18240.394} C_VEL
LIN {X 0,Y 263.137,Z 225.202,A -85,B 0,C 180,E1 -18241.121,E2 -18241.121} C_VEL
LIN {X 0,Y 264.134,Z 227.891,A -85,B 0,C 180,E1 -18241.503,E2 -18241.503} C_VEL
LIN {X 0,Y 266.259,Z 230.015,A -85,B 0,C 180,E1 -18242.145,E2 -18242.145} C_VEL
LIN {X 0,Y 266.917,Z 230.935,A -85,B 0,C 180,E1 -18242.354,E2 -18242.354} C_VEL
LIN {X 0,Y 269.015,Z 234.058,A -85,B 0,C 180,E1 -18243.015,E2 -18243.015} C_VEL
LIN {X 0,Y 270.406,Z 235.792,A -85,B 0,C 180,E1 -18243.429,E2 -18243.429} C_VEL
LIN {X 0,Y 273.148,Z 239.416,A -85,B 0,C 180,E1 -18244.231,E2 -18244.231} C_VEL
LIN {X 0,Y 283.043,Z 253.655,A -85,B 0,C 180,E1 -18246.975,E2 -18246.975} C_VEL
LIN {X 0,Y 292.337,Z 267.835,A -85,B 0,C 180,E1 -18249.333,E2 -18249.333} C_VEL
LIN {X 0,Y 301.428,Z 283.096,A -85,B 0,C 180,E1 -18251.491,E2 -18251.491} C_VEL
LIN {X 0,Y 307.134,Z 293.756,A -85,B 0,C 180,E1 -18252.788,E2 -18252.788} C_VEL
LIN {X 0,Y 305.842,Z 319.925,A -85,B 0,C 180,E1 -18253.42,E2 -18253.42} C_VEL
LIN {X 0,Y 300.485,Z 420.542,A -85,B 0,C 180,E1 -18255.831,E2 -18255.831} C_VEL
LIN {X 0,Y 298.78,Z 437.717,A -85,B 0,C 180,E1 -18256.486,E2 -18256.486} C_VEL
LIN {X 0,Y 296.628,Z 453.622,A -85,B 0,C 180,E1 -18257.344,E2 -18257.344} C_VEL
LIN {X 0,Y 293.915,Z 469.865,A -85,B 0,C 180,E1 -18258.501,E2 -18258.501} C_VEL
LIN {X 0,Y 290.736,Z 485.497,A -85,B 0,C 180,E1 -18259.91,E2 -18259.91} C_VEL
LIN {X 0,Y 287.238,Z 500.291,A -85,B 0,C 180,E1 -18261.562,E2 -18261.562} C_VEL
LIN {X 0,Y 283.483,Z 514.5,A -85,B 0,C 180,E1 -18263.508,E2 -18263.508} C_VEL
LIN {X 0,Y 279.694,Z 527.506,A -85,B 0,C 180,E1 -18265.68,E2 -18265.68} C_VEL
LIN {X 0,Y 276.497,Z 538.144,A -85,B 0,C 180,E1 -18267.819,E2 -18267.819} C_VEL
LIN {X 0,Y 273.045,Z 548.932,A -85,B 0,C 180,E1 -18270.372,E2 -18270.372} C_VEL
LIN {X 0,Y 270.105,Z 558.155,A -85,B 0,C 180,E1 -18272.986,E2 -18272.986} C_VEL
LIN {X 0,Y 267.251,Z 567.036,A -85,B 0,C 180,E1 -18276.042,E2 -18276.042} C_VEL
LIN {X 0,Y 265.082,Z 574.416,A -85,B 0,C 180,E1 -18279.157,E2 -18279.157} C_VEL
LIN {X 0,Y 263.397,Z 580.524,A -85,B 0,C 180,E1 -18282.328,E2 -18282.328} C_VEL
LIN {X 0,Y 262.235,Z 585.384,A -85,B 0,C 180,E1 -18285.549,E2 -18285.549} C_VEL
LIN {X 0,Y 261.363,Z 589.085,A -85,B 0,C 180,E1 -18288.828,E2 -18288.828} C_VEL
LIN {X 0,Y 260.834,Z 591.715,A -85,B 0,C 180,E1 -18292.165,E2 -18292.165} C_VEL
LIN {X 0,Y 260.622,Z 593.179,A -85,B 0,C 180,E1 -18295.563,E2 -18295.563} C_VEL
LIN {X 0,Y 260.7,Z 593.469,A -85,B 0,C 180,E1 -18299.032,E2 -18299.032} C_VEL
LIN {X 0,Y 260.995,Z 592.566,A -85,B 0,C 180,E1 -18302.588,E2 -18302.588} C_VEL
LIN {X 0,Y 261.7,Z 590.263,A -85,B 0,C 180,E1 -18306.325,E2 -18306.325} C_VEL
LIN {X 0,Y 262.886,Z 586.632,A -85,B 0,C 180,E1 -18309.915,E2 -18309.915} C_VEL
LIN {X 0,Y 264.729,Z 581.348,A -85,B 0,C 180,E1 -18313.652,E2 -18313.652} C_VEL
LIN {X 0,Y 266.828,Z 575.613,A -85,B 0,C 180,E1 -18316.778,E2 -18316.778} C_VEL
LIN {X 0,Y 269.495,Z 568.976,A -85,B 0,C 180,E1 -18319.714,E2 -18319.714} C_VEL
LIN {X 0,Y 273.128,Z 559.973,A -85,B 0,C 180,E1 -18322.912,E2 -18322.912} C_VEL
LIN {X 0,Y 276.784,Z 550.692,A -85,B 0,C 180,E1 -18325.615,E2 -18325.615} C_VEL
LIN {X 0,Y 281.235,Z 539.292,A -85,B 0,C 180,E1 -18328.345,E2 -18328.345} C_VEL
LIN {X 0,Y 285.472,Z 527.85,A -85,B 0,C 180,E1 -18330.607,E2 -18330.607} C_VEL
LIN {X 0,Y 289.456,Z 516.238,A -85,B 0,C 180,E1 -18332.527,E2 -18332.527} C_VEL
LIN {X 0,Y 293.658,Z 502.854,A -85,B 0,C 180,E1 -18334.356,E2 -18334.356} C_VEL
LIN {X 0,Y 297.441,Z 489.45,A -85,B 0,C 180,E1 -18335.876,E2 -18335.876} C_VEL
LIN {X 0,Y 301.079,Z 474.848,A -85,B 0,C 180,E1 -18337.229,E2 -18337.229} C_VEL
LIN {X 0,Y 304.318,Z 459.26,A -85,B 0,C 180,E1 -18338.375,E2 -18338.375} C_VEL
LIN {X 0,Y 306.845,Z 443.913,A -85,B 0,C 180,E1 -18339.249,E2 -18339.249} C_VEL
LIN {X 0,Y 308.076,Z 434.622,A -85,B 0,C 180,E1 -18339.674,E2 -18339.674} C_VEL
LIN {X 0,Y 308.302,Z 428.957,A -85,B 0,C 180,E1 -18339.988,E2 -18339.988} C_VEL
LIN {X 0,Y 306.133,Z 410.57,A -85,B 0,C 180,E1 -18341.31,E2 -18341.31} C_VEL
LIN {X 0,Y 306.012,Z 404.805,A -85,B 0,C 180,E1 -18341.555,E2 -18341.555} C_VEL
LIN {X 0,Y 312.721,Z 302.374,A -85,B 0,C 180,E1 -18344.014,E2 -18344.014} C_VEL
LIN {X 0,Y 307.817,Z 293.081,A -85,B 0,C 180,E1 -18345.627,E2 -18345.627} C_VEL
LIN {X 0,Y 300.908,Z 281.553,A -85,B 0,C 180,E1 -18348.086,E2 -18348.086} C_VEL
LIN {X 0,Y 294.81,Z 272.421,A -85,B 0,C 180,E1 -18350.516,E2 -18350.516} C_VEL
LIN {X 0,Y 291.29,Z 267.555,A -85,B 0,C 180,E1 -18352.068,E2 -18352.068} C_VEL
LIN {X 0,Y 288.332,Z 263.36,A -85,B 0,C 180,E1 -18353.517,E2 -18353.517} C_VEL
LIN {X 0,Y 285.491,Z 259.434,A -85,B 0,C 180,E1 -18355.013,E2 -18355.013} C_VEL
LIN {X 0,Y 282.581,Z 255.842,A -85,B 0,C 180,E1 -18356.702,E2 -18356.702} C_VEL
LIN {X 0,Y 281.751,Z 254.671,A -85,B 0,C 180,E1 -18357.238,E2 -18357.238} C_VEL
LIN {X 0,Y 279.107,Z 251.688,A -85,B 0,C 180,E1 -18359.002,E2 -18359.002} C_VEL
LIN {X 0,Y 277.875,Z 249.431,A -85,B 0,C 180,E1 -18359.999,E2 -18359.999} C_VEL
LIN {X 0,Y 275.073,Z 246.903,A -85,B 0,C 180,E1 -18362.379,E2 -18362.379} C_VEL
LIN {X 0,Y 273.425,Z 244.043,A -85,B 0,C 180,E1 -18364.218,E2 -18364.218} C_VEL
LIN {X 0,Y 269.813,Z 241.537,A -85,B 0,C 180,E1 -18370.505,E2 -18370.505} C_VEL
LIN {X 0,Y 269.441,Z 240.993,A -85,B 0,C 180,E1 -18373.576,E2 -18373.576} C_VEL
LIN {X 0,Y 270.166,Z 242.166,A -85,B 0,C 180,E1 -18377.429,E2 -18377.429} C_VEL
LIN {X 0,Y 273.275,Z 244.28,A -85,B 0,C 180,E1 -18382.292,E2 -18382.292} C_VEL
LIN {X 0,Y 274.97,Z 247.469,A -85,B 0,C 180,E1 -18384.231,E2 -18384.231} C_VEL
LIN {X 0,Y 277.77,Z 249.892,A -85,B 0,C 180,E1 -18386.606,E2 -18386.606} C_VEL
LIN {X 0,Y 279.969,Z 253.262,A -85,B 0,C 180,E1 -18388.273,E2 -18388.273} C_VEL
LIN {X 0,Y 282.019,Z 255.332,A -85,B 0,C 180,E1 -18389.589,E2 -18389.589} C_VEL
LIN {X 0,Y 287.175,Z 262.621,A -85,B 0,C 180,E1 -18392.574,E2 -18392.574} C_VEL
LIN {X 0,Y 291.448,Z 269.205,A -85,B 0,C 180,E1 -18394.72,E2 -18394.72} C_VEL
LIN {X 0,Y 295.881,Z 276.306,A -85,B 0,C 180,E1 -18396.684,E2 -18396.684} C_VEL
LIN {X 0,Y 301.609,Z 286.392,A -85,B 0,C 180,E1 -18398.986,E2 -18398.986} C_VEL
LIN {X 0,Y 307.621,Z 298.078,A -85,B 0,C 180,E1 -18401.168,E2 -18401.168} C_VEL
LIN {X 0,Y 312.494,Z 308.824,A -85,B 0,C 180,E1 -18402.821,E2 -18402.821} C_VEL
LIN {X 0,Y 304.197,Z 433.558,A -85,B 0,C 180,E1 -18405.837,E2 -18405.837} C_VEL
LIN {X 0,Y 301.896,Z 451.479,A -85,B 0,C 180,E1 -18406.485,E2 -18406.485} C_VEL
LIN {X 0,Y 298.897,Z 468.298,A -85,B 0,C 180,E1 -18407.351,E2 -18407.351} C_VEL
LIN {X 0,Y 295.834,Z 482.31,A -85,B 0,C 180,E1 -18408.301,E2 -18408.301} C_VEL
LIN {X 0,Y 291.816,Z 498.155,A -85,B 0,C 180,E1 -18409.663,E2 -18409.663} C_VEL
LIN {X 0,Y 287.835,Z 511.663,A -85,B 0,C 180,E1 -18411.086,E2 -18411.086} C_VEL
LIN {X 0,Y 283.604,Z 524.662,A -85,B 0,C 180,E1 -18412.78,E2 -18412.78} C_VEL
LIN {X 0,Y 279.322,Z 536.654,A -85,B 0,C 180,E1 -18414.638,E2 -18414.638} C_VEL
LIN {X 0,Y 275.172,Z 547.749,A -85,B 0,C 180,E1 -18416.691,E2 -18416.691} C_VEL
LIN {X 0,Y 270.827,Z 558.832,A -85,B 0,C 180,E1 -18419.166,E2 -18419.166} C_VEL
LIN {X 0,Y 266.44,Z 569.624,A -85,B 0,C 180,E1 -18422.08,E2 -18422.08} C_VEL
LIN {X 0,Y 263.156,Z 577.72,A -85,B 0,C 180,E1 -18424.7,E2 -18424.7} C_VEL
LIN {X 0,Y 260.157,Z 585.494,A -85,B 0,C 180,E1 -18427.775,E2 -18427.775} C_VEL
LIN {X 0,Y 257.771,Z 591.994,A -85,B 0,C 180,E1 -18430.899,E2 -18430.899} C_VEL
LIN {X 0,Y 256.071,Z 597.354,A -85,B 0,C 180,E1 -18434.067,E2 -18434.067} C_VEL
LIN {X 0,Y 254.862,Z 601.525,A -85,B 0,C 180,E1 -18437.252,E2 -18437.252} C_VEL
LIN {X 0,Y 254.185,Z 604.745,A -85,B 0,C 180,E1 -18440.447,E2 -18440.447} C_VEL
LIN {X 0,Y 253.944,Z 606.866,A -85,B 0,C 180,E1 -18443.641,E2 -18443.641} C_VEL
LIN {X 0,Y 253.937,Z 608.097,A -85,B 0,C 180,E1 -18446.823,E2 -18446.823} C_VEL
LIN {X 0,Y 254.053,Z 608.255,A -85,B 0,C 180,E1 -18449.996,E2 -18449.996} C_VEL
LIN {X 0,Y 253.966,Z 607.506,A -85,B 0,C 180,E1 -18453.169,E2 -18453.169} C_VEL
LIN {X 0,Y 253.941,Z 605.659,A -85,B 0,C 180,E1 -18456.352,E2 -18456.352} C_VEL
LIN {X 0,Y 254.173,Z 602.859,A -85,B 0,C 180,E1 -18459.545,E2 -18459.545} C_VEL
LIN {X 0,Y 255.051,Z 597.799,A -85,B 0,C 180,E1 -18463.541,E2 -18463.541} C_VEL
LIN {X 0,Y 256.205,Z 592.554,A -85,B 0,C 180,E1 -18466.653,E2 -18466.653} C_VEL
LIN {X 0,Y 258.031,Z 585.795,A -85,B 0,C 180,E1 -18469.9,E2 -18469.9} C_VEL
LIN {X 0,Y 260.399,Z 577.963,A -85,B 0,C 180,E1 -18472.983,E2 -18472.983} C_VEL
LIN {X 0,Y 263.461,Z 568.232,A -85,B 0,C 180,E1 -18476.108,E2 -18476.108} C_VEL
LIN {X 0,Y 266.772,Z 558.277,A -85,B 0,C 180,E1 -18478.732,E2 -18478.732} C_VEL
LIN {X 0,Y 270.408,Z 546.613,A -85,B 0,C 180,E1 -18481.314,E2 -18481.314} C_VEL
LIN {X 0,Y 274.396,Z 533.899,A -85,B 0,C 180,E1 -18483.627,E2 -18483.627} C_VEL
LIN {X 0,Y 278.392,Z 520.324,A -85,B 0,C 180,E1 -18485.662,E2 -18485.662} C_VEL
LIN {X 0,Y 281.693,Z 507.718,A -85,B 0,C 180,E1 -18487.224,E2 -18487.224} C_VEL
LIN {X 0,Y 284.841,Z 495.007,A -85,B 0,C 180,E1 -18488.53,E2 -18488.53} C_VEL
LIN {X 0,Y 288.014,Z 479.766,A -85,B 0,C 180,E1 -18489.826,E2 -18489.826} C_VEL
LIN {X 0,Y 290.702,Z 464.135,A -85,B 0,C 180,E1 -18490.857,E2 -18490.857} C_VEL
LIN {X 0,Y 293.064,Z 447.643,A -85,B 0,C 180,E1 -18491.655,E2 -18491.655} C_VEL
LIN {X 0,Y 294.681,Z 431.264,A -85,B 0,C 180,E1 -18492.215,E2 -18492.215} C_VEL
LIN {X 0,Y 301.559,Z 303.874,A -85,B 0,C 180,E1 -18495.302,E2 -18495.302} C_VEL
LIN {X 0,Y 293.193,Z 286.43,A -85,B 0,C 180,E1 -18497.364,E2 -18497.364} C_VEL
LIN {X 0,Y 284.993,Z 271.049,A -85,B 0,C 180,E1 -18499.486,E2 -18499.486} C_VEL
LIN {X 0,Y 276.624,Z 256.708,A -85,B 0,C 180,E1 -18501.795,E2 -18501.795} C_VEL
LIN {X 0,Y 269.118,Z 244.976,A -85,B 0,C 180,E1 -18504.016,E2 -18504.016} C_VEL
LIN {X 0,Y 265.616,Z 239.636,A -85,B 0,C 180,E1 -18505.113,E2 -18505.113} C_VEL
LIN {X 0,Y 262.908,Z 235.822,A -85,B 0,C 180,E1 -18505.982,E2 -18505.982} C_VEL
LIN {X 0,Y 260.601,Z 233.124,A -85,B 0,C 180,E1 -18506.719,E2 -18506.719} C_VEL
LIN {X 0,Y 259.533,Z 231.125,A -85,B 0,C 180,E1 -18507.102,E2 -18507.102} C_VEL
LIN {X 0,Y 257.231,Z 228.986,A -85,B 0,C 180,E1 -18507.846,E2 -18507.846} C_VEL
LIN {X 0,Y 256.193,Z 226.605,A -85,B 0,C 180,E1 -18508.259,E2 -18508.259} C_VEL
LIN {X 0,Y 256.066,Z 225.875,A -85,B 0,C 180,E1 -18508.338,E2 -18508.338} C_VEL
LIN {X 0,Y 256.116,Z 225.876,A -85,B 0,C 180,E1 -18512.194,E2 -18512.194} C_VEL
LIN {X 0,Y 256.148,Z 225.879,A -85,B 0,C 180,E1 -18515.698,E2 -18515.698} C_VEL
LIN {X 0,Y 256.211,Z 225.851,A -85,B 0,C 180,E1 -18519.11,E2 -18519.11} C_VEL
LIN {X 0,Y 256.268,Z 225.876,A -85,B 0,C 180,E1 -18524.084,E2 -18524.084} C_VEL
LIN {X 0,Y 256.283,Z 225.831,A -85,B 0,C 180,E1 -18528.934,E2 -18528.934} C_VEL
LIN {X 0,Y 256.511,Z 225.846,A -85,B 0,C 180,E1 -18532.127,E2 -18532.127} C_VEL
LIN {X 0,Y 256.687,Z 225.789,A -85,B 0,C 180,E1 -18538.432,E2 -18538.432} C_VEL
LIN {X 0,Y 256.687,Z 225.822,A -85,B 0,C 180,E1 -18541.57,E2 -18541.57} C_VEL
LIN {X 0,Y 256.443,Z 225.839,A -85,B 0,C 180,E1 -18546.794,E2 -18546.794} C_VEL
LIN {X 0,Y 256.402,Z 225.847,A -85,B 0,C 180,E1 -18549.467,E2 -18549.467} C_VEL
LIN {X 0,Y 256.225,Z 225.873,A -85,B 0,C 180,E1 -18554.293,E2 -18554.293} C_VEL
LIN {X 0,Y 256.186,Z 225.86,A -85,B 0,C 180,E1 -18557.565,E2 -18557.565} C_VEL
LIN {X 0,Y 256.134,Z 225.88,A -85,B 0,C 180,E1 -18561.122,E2 -18561.122} C_VEL
LIN {X 0,Y 256.166,Z 225.86,A -85,B 0,C 180,E1 -18565.141,E2 -18565.141} C_VEL
LIN {X 0,Y 256.093,Z 225.898,A -85,B 0,C 180,E1 -18569.603,E2 -18569.603} C_VEL
LIN {X 0,Y 256.049,Z 225.875,A -85,B 0,C 180,E1 -18573.297,E2 -18573.297} C_VEL
LIN {X 0,Y 256.096,Z 225.889,A -85,B 0,C 180,E1 -18577.274,E2 -18577.274} C_VEL
